C09125=1232.862,309.297,-67.480,-176.248,6.770,148.147
C09126=1232.866,309.049,-67.449,-176.251,6.767,148.147
C09127=1232.870,308.801,-67.420,-176.253,6.765,148.147
C09128=1232.875,308.552,-67.390,-176.255,6.763,148.147
C09129=1232.880,308.304,-67.361,-176.257,6.760,148.147
C09130=1232.884,308.056,-67.331,-176.260,6.757,148.147
C09131=1232.888,307.808,-67.301,-176.262,6.755,148.148
C09132=1232.892,307.560,-67.271,-176.264,6.753,148.148
C09133=1232.897,307.311,-67.241,-176.266,6.751,148.148
C09134=1232.901,307.063,-67.212,-176.269,6.748,148.148
C09135=1232.905,306.815,-67.182,-176.271,6.746,148.148
C09136=1232.909,306.566,-67.153,-176.273,6.743,148.148
C09137=1232.913,306.318,-67.124,-176.275,6.741,148.148
C09138=1232.918,306.070,-67.094,-176.278,6.739,148.148
C09139=1232.923,305.821,-67.064,-176.280,6.736,148.148
C09140=1232.926,305.574,-67.034,-176.282,6.734,148.148
C09141=1232.931,305.325,-67.004,-176.284,6.732,148.148
C09142=1232.935,305.077,-66.975,-176.286,6.729,148.148
C09143=1232.940,304.830,-66.946,-176.289,6.726,148.148
C09144=1232.944,304.581,-66.916,-176.291,6.724,148.148
C09145=1232.948,304.333,-66.887,-176.293,6.722,148.148
C09146=1232.952,304.085,-66.858,-176.295,6.720,148.148
C09147=1232.956,303.837,-66.828,-176.298,6.718,148.149
C09148=1232.960,303.588,-66.799,-176.301,6.715,148.149
C09149=1232.965,303.340,-66.769,-176.303,6.712,148.149
C09150=1232.970,303.091,-66.739,-176.305,6.710,148.149
C09151=1232.974,302.843,-66.710,-176.307,6.708,148.149
C09152=1232.979,302.595,-66.681,-176.310,6.705,148.149
C09153=1232.983,302.347,-66.652,-176.312,6.703,148.149
C09154=1232.987,302.098,-66.622,-176.314,6.700,148.149
C09155=1232.991,301.850,-66.593,-176.316,6.698,148.149
C09156=1232.996,301.602,-66.564,-176.319,6.696,148.149
C09157=1233.000,301.354,-66.534,-176.321,6.693,148.149
C09158=1233.004,301.105,-66.505,-176.323,6.691,148.149
C09159=1233.009,300.858,-66.476,-176.325,6.689,148.149
C09160=1233.013,300.610,-66.446,-176.327,6.687,148.149
C09161=1233.017,300.361,-66.417,-176.331,6.684,148.150
C09162=1233.022,300.112,-66.388,-176.333,6.682,148.150
C09163=1233.026,299.864,-66.358,-176.335,6.679,148.150
C09164=1233.031,299.617,-66.329,-176.337,6.677,148.150
C09165=1233.035,299.368,-66.300,-176.339,6.675,148.150
C09166=1233.039,299.119,-66.271,-176.342,6.672,148.150
C09167=1233.043,298.871,-66.242,-176.344,6.670,148.150
C09168=1233.047,298.623,-66.213,-176.346,6.668,148.150
C09169=1233.051,298.375,-66.183,-176.348,6.665,148.150
C09170=1233.056,298.127,-66.155,-176.351,6.663,148.150
C09171=1233.060,297.878,-66.126,-176.354,6.660,148.151
C09172=1233.064,297.630,-66.096,-176.356,6.658,148.151
C09173=1233.069,297.381,-66.067,-176.358,6.656,148.151
C09174=1233.074,297.134,-66.038,-176.360,6.654,148.151
C09175=1233.078,296.885,-66.009,-176.362,6.652,148.151
C09176=1233.082,296.637,-65.979,-176.365,6.649,148.151
C09177=1233.086,296.389,-65.951,-176.367,6.647,148.151
C09178=1233.090,296.140,-65.922,-176.369,6.644,148.151
C09179=1233.095,295.892,-65.893,-176.372,6.642,148.151
C09180=1233.099,295.644,-65.864,-176.374,6.640,148.151
C09181=1233.103,295.396,-65.834,-176.377,6.637,148.151
C09182=1233.108,295.147,-65.806,-176.379,6.635,148.152
C09183=1233.112,294.899,-65.777,-176.381,6.633,148.152
C09184=1233.116,294.651,-65.749,-176.384,6.631,148.152
C09185=1233.121,294.402,-65.719,-176.386,6.629,148.152
C09186=1233.125,294.155,-65.690,-176.388,6.626,148.152
C09187=1233.130,293.906,-65.661,-176.390,6.623,148.152
C09188=1233.133,293.658,-65.632,-176.393,6.621,148.152
C09189=1233.138,293.409,-65.604,-176.395,6.619,148.152
C09190=1233.143,293.161,-65.575,-176.397,6.617,148.152
C09191=1233.147,292.913,-65.546,-176.400,6.614,148.153
C09192=1233.151,292.665,-65.517,-176.402,6.612,148.153
C09193=1233.156,292.416,-65.489,-176.405,6.610,148.153
C09194=1233.160,292.168,-65.459,-176.407,6.608,148.153
C09195=1233.164,291.919,-65.430,-176.409,6.606,148.153
C09196=1233.169,291.671,-65.403,-176.411,6.603,148.153
C09197=1233.173,291.423,-65.373,-176.414,6.600,148.153
C09198=1233.177,291.174,-65.344,-176.417,6.598,148.153
C09199=1233.181,290.927,-65.316,-176.419,6.596,148.154
C09200=1233.186,290.678,-65.287,-176.421,6.594,148.154
C09201=1233.190,290.430,-65.258,-176.423,6.592,148.154
C09202=1233.195,290.182,-65.229,-176.426,6.590,148.154
C09203=1233.199,289.908,-65.198,-176.429,6.587,148.154
C09204=1233.204,289.633,-65.167,-176.431,6.585,148.154
C09205=1233.209,289.359,-65.135,-176.434,6.582,148.154
C09206=1233.214,289.086,-65.103,-176.436,6.580,148.155
C09207=1233.218,288.837,-65.074,-176.439,6.577,148.155
C09208=1233.222,288.588,-65.046,-176.441,6.575,148.155
C09209=1233.227,288.341,-65.017,-176.443,6.573,148.155
C09210=1233.231,288.092,-64.988,-176.445,6.571,148.155
C09211=1233.235,287.843,-64.960,-176.448,6.569,148.155
C09212=1233.240,287.595,-64.932,-176.450,6.566,148.155
C09213=1233.244,287.347,-64.903,-176.453,6.564,148.156
C09214=1233.249,287.099,-64.875,-176.455,6.561,148.156
C09215=1233.253,286.850,-64.846,-176.457,6.559,148.156
C09216=1233.257,286.602,-64.818,-176.460,6.557,148.156
C09217=1233.262,286.353,-64.789,-176.462,6.555,148.156
C09218=1233.266,286.105,-64.760,-176.465,6.553,148.156
C09219=1233.271,285.857,-64.732,-176.467,6.550,148.156
C09220=1233.274,285.609,-64.704,-176.470,6.548,148.156
C09221=1233.280,285.360,-64.676,-176.472,6.546,148.157
C09222=1233.283,285.112,-64.647,-176.474,6.544,148.157
C09223=1233.288,284.864,-64.619,-176.477,6.542,148.157
C09224=1233.293,284.615,-64.590,-176.479,6.540,148.157
C09225=1233.296,284.367,-64.562,-176.481,6.537,148.157
C09226=1233.301,284.119,-64.533,-176.484,6.535,148.157
C09227=1233.305,283.870,-64.505,-176.486,6.532,148.157
C09228=1233.310,283.622,-64.477,-176.489,6.531,148.158
C09229=1233.314,283.373,-64.448,-176.491,6.528,148.158
C09230=1233.318,283.125,-64.421,-176.494,6.526,148.158
C09231=1233.323,282.877,-64.392,-176.496,6.524,148.158
C09232=1233.327,282.629,-64.364,-176.498,6.522,148.158
C09233=1233.332,282.380,-64.335,-176.501,6.519,148.158
C09234=1233.336,282.132,-64.308,-176.503,6.517,148.158
C09235=1233.340,281.883,-64.279,-176.506,6.515,148.159
C09236=1233.345,281.635,-64.251,-176.508,6.513,148.159
C09237=1233.349,281.386,-64.222,-176.510,6.511,148.159
C09238=1233.354,281.138,-64.195,-176.512,6.509,148.159
C09239=1233.357,280.890,-64.166,-176.515,6.507,148.159
C09240=1233.363,280.642,-64.138,-176.517,6.505,148.160
C09241=1233.366,280.393,-64.110,-176.520,6.502,148.160
C09242=1233.371,280.145,-64.082,-176.522,6.500,148.160
C09243=1233.375,279.896,-64.053,-176.525,6.498,148.160
C09244=1233.379,279.648,-64.026,-176.527,6.496,148.160
C09245=1233.384,279.400,-63.997,-176.530,6.494,148.161
C09246=1233.389,279.151,-63.970,-176.532,6.491,148.161
C09247=1233.392,278.902,-63.942,-176.534,6.489,148.161
C09248=1233.397,278.654,-63.913,-176.536,6.487,148.161
C09249=1233.402,278.406,-63.886,-176.539,6.485,148.161
C09250=1233.406,278.158,-63.857,-176.542,6.482,148.161
C09251=1233.411,277.910,-63.829,-176.544,6.480,148.161
C09252=1233.414,277.661,-63.801,-176.546,6.478,148.162
C09253=1233.419,277.413,-63.774,-176.549,6.476,148.162
C09254=1233.424,277.164,-63.745,-176.551,6.474,148.162
C09255=1233.428,276.916,-63.717,-176.554,6.472,148.162
C09256=1233.432,276.668,-63.690,-176.556,6.470,148.162
C09257=1233.436,276.419,-63.662,-176.558,6.468,148.163
C09258=1233.441,276.171,-63.634,-176.561,6.466,148.163
C09259=1233.445,275.922,-63.606,-176.564,6.463,148.163
C09260=1233.449,275.674,-63.578,-176.566,6.461,148.163
C09261=1233.454,275.426,-63.551,-176.568,6.459,148.163
C09262=1233.459,275.177,-63.522,-176.571,6.457,148.163
C09263=1233.463,274.929,-63.494,-176.573,6.455,148.164
C09264=1233.467,274.680,-63.467,-176.575,6.453,148.164
C09265=1233.471,274.432,-63.439,-176.578,6.451,148.164
C09266=1233.476,274.184,-63.411,-176.580,6.449,148.164
C09267=1233.480,273.934,-63.383,-176.583,6.447,148.164
C09268=1233.485,273.687,-63.356,-176.585,6.445,148.165
C09269=1233.489,273.439,-63.328,-176.588,6.442,148.165
C09270=1233.493,273.189,-63.300,-176.590,6.440,148.165
C09271=1233.498,272.941,-63.272,-176.592,6.438,148.165
C09272=1233.503,272.693,-63.245,-176.595,6.436,148.165
C09273=1233.507,272.444,-63.217,-176.597,6.433,148.165
C09274=1233.511,272.196,-63.189,-176.600,6.432,148.166
C09275=1233.516,271.948,-63.162,-176.602,6.430,148.166
C09276=1233.520,271.699,-63.134,-176.604,6.427,148.166
C09277=1233.524,271.451,-63.107,-176.607,6.426,148.166
C09278=1233.529,271.203,-63.078,-176.609,6.423,148.166
C09279=1233.533,270.953,-63.051,-176.612,6.421,148.167
C09280=1233.538,270.705,-63.023,-176.614,6.419,148.167
C09281=1233.542,270.457,-62.996,-176.617,6.417,148.167
C09282=1233.546,270.208,-62.968,-176.620,6.415,148.167
C09283=1233.551,269.960,-62.941,-176.622,6.412,148.167
C09284=1233.555,269.712,-62.913,-176.624,6.410,148.168
C09285=1233.559,269.463,-62.886,-176.626,6.408,148.168
C09286=1233.564,269.214,-62.859,-176.629,6.406,148.168
C09287=1233.568,268.966,-62.831,-176.632,6.404,148.168
C09288=1233.573,268.718,-62.804,-176.634,6.402,148.168
C09289=1233.577,268.469,-62.776,-176.636,6.400,148.169
C09290=1233.581,268.221,-62.749,-176.639,6.398,148.169
C09291=1233.586,267.973,-62.721,-176.641,6.396,148.169
C09292=1233.591,267.724,-62.693,-176.644,6.394,148.169
C09293=1233.595,267.475,-62.666,-176.646,6.392,148.169
C09294=1233.599,267.227,-62.638,-176.648,6.390,148.170
C09295=1233.604,266.979,-62.611,-176.651,6.388,148.170
C09296=1233.609,266.730,-62.584,-176.653,6.386,148.170
C09297=1233.612,266.482,-62.556,-176.656,6.384,148.170
C09298=1233.617,266.233,-62.529,-176.658,6.382,148.171
C09299=1233.621,265.985,-62.502,-176.660,6.380,148.171
C09300=1233.626,265.736,-62.475,-176.664,6.377,148.171
C09301=1233.630,265.489,-62.447,-176.666,6.375,148.171
C09302=1233.634,265.239,-62.420,-176.668,6.373,148.171
C09303=1233.639,264.991,-62.393,-176.671,6.371,148.172
C09304=1233.643,264.742,-62.366,-176.673,6.369,148.172
C09305=1233.648,264.494,-62.338,-176.676,6.367,148.172
C09306=1233.652,264.246,-62.311,-176.678,6.365,148.172
C09307=1233.657,263.973,-62.280,-176.681,6.363,148.173
C09308=1233.662,263.700,-62.251,-176.683,6.361,148.173
C09309=1233.666,263.427,-62.221,-176.686,6.358,148.173
C09310=1233.672,263.155,-62.191,-176.689,6.357,148.173
C09311=1233.676,262.906,-62.164,-176.691,6.355,148.174
C09312=1233.680,262.658,-62.138,-176.693,6.352,148.174
C09313=1233.685,262.410,-62.110,-176.696,6.351,148.174
C09314=1233.689,262.162,-62.083,-176.699,6.349,148.174
C09315=1233.693,261.913,-62.055,-176.701,6.347,148.175
C09316=1233.698,261.664,-62.028,-176.703,6.345,148.175
C09317=1233.703,261.416,-62.001,-176.706,6.343,148.175
C09318=1233.707,261.167,-61.974,-176.709,6.341,148.175
C09319=1233.711,260.919,-61.948,-176.711,6.339,148.175
C09320=1233.716,260.670,-61.921,-176.713,6.337,148.176
C09321=1233.720,260.422,-61.894,-176.716,6.335,148.176
C09322=1233.725,260.173,-61.867,-176.718,6.333,148.176
C09323=1233.729,259.924,-61.839,-176.721,6.331,148.176
C09324=1233.733,259.676,-61.813,-176.723,6.329,148.177
C09325=1233.738,259.427,-61.786,-176.726,6.327,148.177
C09326=1233.742,259.179,-61.759,-176.728,6.325,148.177
C09327=1233.747,258.931,-61.731,-176.730,6.323,148.177
C09328=1233.751,258.682,-61.705,-176.733,6.321,148.178
C09329=1233.756,258.434,-61.678,-176.735,6.319,148.178
C09330=1233.760,258.185,-61.651,-176.738,6.317,148.178
C09331=1233.765,257.937,-61.624,-176.740,6.315,148.178
C09332=1233.769,257.689,-61.597,-176.743,6.313,148.179
C09333=1233.773,257.439,-61.570,-176.745,6.311,148.179
C09334=1233.778,257.191,-61.543,-176.748,6.309,148.179
C09335=1233.782,256.942,-61.516,-176.750,6.307,148.179
C09336=1233.786,256.694,-61.489,-176.753,6.305,148.180
C09337=1233.791,256.445,-61.463,-176.755,6.303,148.180
C09338=1233.796,256.197,-61.436,-176.758,6.301,148.180
C09339=1233.800,255.948,-61.409,-176.760,6.299,148.180
C09340=1233.804,255.700,-61.382,-176.763,6.297,148.181
C09341=1233.809,255.451,-61.355,-176.765,6.295,148.181
C09342=1233.813,255.203,-61.329,-176.768,6.293,148.181
C09343=1233.818,254.954,-61.303,-176.770,6.291,148.181
C09344=1233.823,254.706,-61.275,-176.773,6.289,148.182
C09345=1233.827,254.458,-61.249,-176.775,6.287,148.182
C09346=1233.831,254.209,-61.222,-176.778,6.285,148.182
C09347=1233.836,253.960,-61.196,-176.780,6.283,148.182
C09348=1233.840,253.712,-61.169,-176.783,6.281,148.183
C09349=1233.845,253.463,-61.142,-176.785,6.279,148.183
C09350=1233.849,253.215,-61.116,-176.787,6.277,148.183
C09351=1233.854,252.966,-61.089,-176.790,6.275,148.183
C09352=1233.858,252.717,-61.062,-176.793,6.274,148.184
C09353=1233.862,252.469,-61.036,-176.795,6.271,148.184
C09354=1233.867,252.221,-61.009,-176.797,6.269,148.184
C09355=1233.871,251.972,-60.983,-176.800,6.268,148.184
C09356=1233.876,251.723,-60.956,-176.803,6.266,148.185
C09357=1233.880,251.475,-60.929,-176.805,6.264,148.185
C09358=1233.885,251.226,-60.903,-176.807,6.262,148.185
C09359=1233.888,250.978,-60.877,-176.810,6.260,148.185
C09360=1233.893,250.729,-60.850,-176.813,6.258,148.186
C09361=1233.897,250.481,-60.824,-176.815,6.256,148.186
C09362=1233.902,250.232,-60.797,-176.818,6.254,148.186
C09363=1233.906,249.983,-60.771,-176.820,6.252,148.186
C09364=1233.911,249.735,-60.744,-176.822,6.250,148.187
C09365=1233.915,249.486,-60.718,-176.825,6.249,148.187
C09366=1233.920,249.238,-60.691,-176.827,6.247,148.187
C09367=1233.925,248.989,-60.666,-176.830,6.245,148.188
C09368=1233.929,248.741,-60.639,-176.832,6.243,148.188
C09369=1233.934,248.492,-60.613,-176.834,6.241,148.188
C09370=1233.938,248.244,-60.586,-176.837,6.239,148.188
C09371=1233.942,247.995,-60.560,-176.840,6.237,148.189
C09372=1233.947,247.746,-60.533,-176.842,6.235,148.189
C09373=1233.951,247.498,-60.507,-176.844,6.233,148.189
C09374=1233.956,247.249,-60.480,-176.847,6.231,148.189
C09375=1233.960,247.000,-60.454,-176.850,6.229,148.190
C09376=1233.964,246.752,-60.428,-176.852,6.227,148.190
C09377=1233.970,246.504,-60.402,-176.855,6.226,148.190
C09378=1233.974,246.255,-60.376,-176.857,6.224,148.191
C09379=1233.979,246.006,-60.349,-176.860,6.221,148.191
C09380=1233.982,245.758,-60.323,-176.862,6.220,148.191
C09381=1233.987,245.509,-60.297,-176.865,6.218,148.191
C09382=1233.992,245.260,-60.271,-176.867,6.217,148.192
C09383=1233.996,245.012,-60.244,-176.869,6.215,148.192
C09384=1234.000,244.764,-60.219,-176.872,6.213,148.192
C09385=1234.005,244.515,-60.192,-176.875,6.211,148.193
C09386=1234.009,244.267,-60.166,-176.877,6.209,148.193
C09387=1234.013,244.018,-60.140,-176.879,6.207,148.193
C09388=1234.018,243.769,-60.114,-176.882,6.205,148.193
C09389=1234.022,243.521,-60.087,-176.885,6.203,148.194
C09390=1234.027,243.272,-60.062,-176.887,6.201,148.194
C09391=1234.032,243.023,-60.036,-176.890,6.199,148.194
C09392=1234.036,242.775,-60.009,-176.892,6.197,148.194
C09393=1234.040,242.526,-59.983,-176.895,6.195,148.195
C09394=1234.045,242.277,-59.957,-176.897,6.194,148.195
C09395=1234.049,242.028,-59.931,-176.899,6.192,148.195
C09396=1234.054,241.780,-59.906,-176.902,6.190,148.196
C09397=1234.058,241.532,-59.879,-176.905,6.189,148.196
C09398=1234.063,241.283,-59.853,-176.907,6.187,148.196
C09399=1234.067,241.034,-59.827,-176.910,6.185,148.196
C09400=1234.072,240.785,-59.802,-176.912,6.183,148.197
C09401=1234.076,240.537,-59.776,-176.914,6.181,148.197
C09402=1234.081,240.289,-59.749,-176.917,6.179,148.197
C09403=1234.085,240.040,-59.723,-176.920,6.177,148.198
C09404=1234.090,239.791,-59.698,-176.922,6.175,148.198
C09405=1234.094,239.543,-59.672,-176.924,6.174,148.198
C09406=1234.099,239.294,-59.646,-176.927,6.172,148.199
C09407=1234.104,239.045,-59.620,-176.930,6.170,148.199
C09408=1234.108,238.796,-59.594,-176.932,6.168,148.199
C09409=1234.112,238.549,-59.568,-176.934,6.166,148.199
C09410=1234.117,238.300,-59.543,-176.937,6.164,148.200
C09411=1234.121,238.028,-59.515,-176.940,6.162,148.200
C09412=1234.127,237.757,-59.487,-176.943,6.161,148.200
C09413=1234.131,237.486,-59.458,-176.945,6.159,148.201
C09414=1234.136,237.215,-59.430,-176.948,6.156,148.201
C09415=1234.141,236.965,-59.404,-176.951,6.155,148.201
C09416=1234.145,236.717,-59.378,-176.953,6.153,148.202
C09417=1234.150,236.469,-59.353,-176.955,6.151,148.202
C09418=1234.154,236.220,-59.327,-176.958,6.149,148.202
C09419=1234.159,235.971,-59.301,-176.960,6.147,148.202
C09420=1234.163,235.722,-59.276,-176.963,6.145,148.203
C09421=1234.168,235.474,-59.250,-176.966,6.143,148.203
C09422=1234.172,235.225,-59.225,-176.968,6.142,148.203
C09423=1234.176,234.976,-59.199,-176.970,6.141,148.204
C09424=1234.181,234.728,-59.173,-176.973,6.139,148.204
C09425=1234.186,234.479,-59.147,-176.976,6.137,148.204
C09426=1234.190,234.230,-59.122,-176.978,6.135,148.205
C09427=1234.195,233.982,-59.097,-176.981,6.133,148.205
C09428=1234.200,233.733,-59.071,-176.983,6.131,148.205
C09429=1234.204,233.484,-59.045,-176.986,6.129,148.206
C09430=1234.209,233.236,-59.020,-176.989,6.127,148.206
C09431=1234.213,232.987,-58.994,-176.990,6.126,148.206
C09432=1234.217,232.738,-58.968,-176.993,6.124,148.206
C09433=1234.222,232.490,-58.944,-176.996,6.122,148.207
C09434=1234.226,232.241,-58.918,-176.998,6.120,148.207
C09435=1234.231,231.993,-58.893,-177.001,6.119,148.207
C09436=1234.235,231.744,-58.867,-177.003,6.117,148.208
C09437=1234.240,231.495,-58.841,-177.006,6.115,148.208
C09438=1234.245,231.246,-58.816,-177.008,6.114,148.208
C09439=1234.249,230.998,-58.791,-177.011,6.112,148.209
C09440=1234.254,230.749,-58.765,-177.013,6.110,148.209
C09441=1234.258,230.501,-58.739,-177.016,6.108,148.209
C09442=1234.262,230.252,-58.715,-177.019,6.106,148.210
C09443=1234.267,230.003,-58.690,-177.021,6.104,148.210
C09444=1234.271,229.755,-58.664,-177.024,6.102,148.210
C09445=1234.276,229.507,-58.638,-177.026,6.101,148.211
C09446=1234.280,229.257,-58.613,-177.028,6.100,148.211
C09447=1234.285,229.008,-58.588,-177.031,6.098,148.211
C09448=1234.289,228.760,-58.562,-177.034,6.096,148.212
C09449=1234.294,228.511,-58.537,-177.036,6.094,148.212
C09450=1234.299,228.263,-58.512,-177.039,6.092,148.212
C09451=1234.303,228.014,-58.486,-177.041,6.091,148.213
C09452=1234.308,227.765,-58.461,-177.044,6.089,148.213
C09453=1234.312,227.517,-58.436,-177.046,6.087,148.213
C09454=1234.316,227.267,-58.411,-177.049,6.085,148.214
C09455=1234.321,227.019,-58.386,-177.051,6.083,148.214
C09456=1234.325,226.770,-58.360,-177.054,6.082,148.214
C09457=1234.330,226.522,-58.335,-177.057,6.080,148.214
C09458=1234.334,226.273,-58.310,-177.059,6.079,148.215
C09459=1234.339,226.024,-58.286,-177.061,6.077,148.215
C09460=1234.343,225.776,-58.260,-177.064,6.075,148.216
C09461=1234.348,225.527,-58.235,-177.067,6.073,148.216
C09462=1234.352,225.278,-58.209,-177.069,6.071,148.216
C09463=1234.358,225.029,-58.185,-177.072,6.069,148.216
C09464=1234.361,224.781,-58.160,-177.074,6.068,148.217
C09465=1234.366,224.532,-58.135,-177.077,6.066,148.217
C09466=1234.370,224.283,-58.109,-177.079,6.064,148.217
C09467=1234.376,224.035,-58.085,-177.082,6.063,148.218
C09468=1234.379,223.786,-58.059,-177.084,6.061,148.218
C09469=1234.384,223.537,-58.035,-177.086,6.060,148.218
C09470=1234.388,223.289,-58.009,-177.089,6.058,148.219
C09471=1234.394,223.040,-57.984,-177.092,6.056,148.219
C09472=1234.397,222.791,-57.959,-177.094,6.054,148.219
C09473=1234.402,222.543,-57.934,-177.097,6.052,148.220
C09474=1234.407,222.294,-57.910,-177.100,6.050,148.220
C09475=1234.411,222.045,-57.884,-177.102,6.049,148.220
C09476=1234.416,221.797,-57.860,-177.104,6.047,148.221
C09477=1234.420,221.547,-57.835,-177.107,6.046,148.221
C09478=1234.425,221.299,-57.810,-177.110,6.044,148.221
C09479=1234.429,221.050,-57.785,-177.112,6.042,148.222
C09480=1234.434,220.802,-57.760,-177.114,6.041,148.222
C09481=1234.438,220.552,-57.735,-177.117,6.039,148.222
C09482=1234.443,220.304,-57.711,-177.119,6.037,148.223
C09483=1234.448,220.055,-57.686,-177.122,6.035,148.223
C09484=1234.452,219.807,-57.660,-177.125,6.033,148.223
C09485=1234.457,219.558,-57.636,-177.127,6.031,148.224
C09486=1234.461,219.309,-57.611,-177.129,6.030,148.224
C09487=1234.465,219.061,-57.586,-177.132,6.028,148.224
C09488=1234.470,218.812,-57.562,-177.135,6.027,148.225
C09489=1234.475,218.563,-57.537,-177.138,6.025,148.225
C09490=1234.479,218.314,-57.513,-177.140,6.023,148.226
C09491=1234.484,218.065,-57.488,-177.142,6.022,148.226
C09492=1234.488,217.817,-57.463,-177.145,6.020,148.226
C09493=1234.493,217.568,-57.438,-177.148,6.018,148.227
C09494=1234.498,217.319,-57.413,-177.150,6.017,148.227
C09495=1234.502,217.071,-57.389,-177.153,6.015,148.227
C09496=1234.506,216.821,-57.364,-177.155,6.014,148.228
C09497=1234.511,216.573,-57.339,-177.158,6.012,148.228
C09498=1234.516,216.325,-57.314,-177.160,6.010,148.228
C09499=1234.519,216.076,-57.290,-177.163,6.008,148.229
C09500=1234.525,215.827,-57.265,-177.166,6.006,148.229
C09501=1234.529,215.578,-57.241,-177.168,6.005,148.229
C09502=1234.533,215.329,-57.216,-177.170,6.003,148.230
C09503=1234.538,215.081,-57.192,-177.173,6.002,148.230
C09504=1234.543,214.832,-57.167,-177.176,6.000,148.231
C09505=1234.547,214.583,-57.143,-177.179,5.998,148.231
C09506=1234.552,214.334,-57.118,-177.181,5.997,148.231
C09507=1234.556,214.086,-57.094,-177.183,5.995,148.232
C09508=1234.561,213.837,-57.069,-177.186,5.993,148.232
C09509=1234.565,213.588,-57.044,-177.189,5.991,148.232
C09510=1234.570,213.340,-57.020,-177.191,5.990,148.233
C09511=1234.574,213.091,-56.996,-177.193,5.988,148.233
C09512=1234.579,212.842,-56.971,-177.196,5.987,148.233
C09513=1234.583,212.593,-56.947,-177.198,5.985,148.234
C09514=1234.589,212.345,-56.922,-177.202,5.983,148.234
C09515=1234.593,212.073,-56.896,-177.204,5.981,148.235
C09516=1234.598,211.803,-56.869,-177.207,5.979,148.235
C09517=1234.603,211.533,-56.843,-177.209,5.978,148.235
C09518=1234.608,211.263,-56.816,-177.213,5.976,148.236
C09519=1234.613,211.014,-56.793,-177.215,5.975,148.236
C09520=1234.617,210.764,-56.768,-177.217,5.973,148.236
C09521=1234.622,210.516,-56.744,-177.220,5.971,148.237
C09522=1234.626,210.268,-56.720,-177.223,5.969,148.237
C09523=1234.631,210.019,-56.695,-177.225,5.968,148.238
C09524=1234.635,209.770,-56.670,-177.227,5.966,148.238
C09525=1234.640,209.521,-56.646,-177.230,5.965,148.238
C09526=1234.645,209.273,-56.622,-177.233,5.963,148.239
C09527=1234.649,209.024,-56.598,-177.235,5.962,148.239
C09528=1234.654,208.774,-56.573,-177.238,5.960,148.239
C09529=1234.658,208.526,-56.549,-177.240,5.958,148.240
C09530=1234.663,208.277,-56.525,-177.243,5.956,148.240
C09531=1234.668,208.029,-56.500,-177.245,5.955,148.240
C09532=1234.672,207.780,-56.477,-177.248,5.954,148.241
C09533=1234.676,207.531,-56.453,-177.251,5.952,148.241
C09534=1234.681,207.282,-56.429,-177.253,5.950,148.242
C09535=1234.686,207.033,-56.404,-177.255,5.949,148.242
C09536=1234.690,206.784,-56.381,-177.258,5.947,148.242
C09537=1234.695,206.536,-56.356,-177.261,5.945,148.243
C09538=1234.699,206.287,-56.331,-177.263,5.944,148.243
C09539=1234.704,206.038,-56.307,-177.265,5.942,148.243
C09540=1234.708,205.789,-56.284,-177.268,5.941,148.244
C09541=1234.713,205.541,-56.260,-177.271,5.939,148.244
C09542=1234.718,205.292,-56.235,-177.273,5.938,148.245
C09543=1234.723,205.043,-56.212,-177.276,5.936,148.245
C09544=1234.726,204.794,-56.187,-177.279,5.934,148.245
C09545=1234.731,204.545,-56.163,-177.281,5.932,148.246
C09546=1234.736,204.296,-56.140,-177.283,5.931,148.246
C09547=1234.741,204.048,-56.115,-177.286,5.930,148.246
C09548=1234.745,203.799,-56.092,-177.289,5.928,148.247
C09549=1234.750,203.550,-56.068,-177.291,5.927,148.247
C09550=1234.754,203.302,-56.044,-177.294,5.925,148.248
C09551=1234.758,203.052,-56.020,-177.296,5.923,148.248
C09552=1234.763,202.804,-55.996,-177.299,5.921,148.248
C09553=1234.768,202.554,-55.972,-177.301,5.920,148.249
C09554=1234.773,202.306,-55.948,-177.304,5.919,148.249
C09555=1234.777,202.057,-55.924,-177.307,5.917,148.250
C09556=1234.782,201.808,-55.901,-177.309,5.916,148.250
C09557=1234.786,201.560,-55.877,-177.312,5.914,148.250
C09558=1234.791,201.311,-55.853,-177.314,5.912,148.251
C09559=1234.795,201.063,-55.829,-177.316,5.911,148.251
C09560=1234.800,200.813,-55.805,-177.319,5.910,148.252
C09561=1234.804,200.564,-55.781,-177.322,5.908,148.252
C09562=1234.809,200.315,-55.757,-177.325,5.906,148.252
C09563=1234.814,200.066,-55.734,-177.327,5.905,148.253
C09564=1234.818,199.818,-55.710,-177.329,5.903,148.253
C09565=1234.823,199.569,-55.687,-177.332,5.901,148.253
C09566=1234.827,199.320,-55.662,-177.335,5.900,148.254
C09567=1234.832,199.071,-55.639,-177.337,5.899,148.254
C09568=1234.836,198.823,-55.615,-177.340,5.897,148.255
C09569=1234.841,198.574,-55.592,-177.342,5.896,148.255
C09570=1234.846,198.325,-55.568,-177.345,5.894,148.255
C09571=1234.850,198.076,-55.544,-177.348,5.892,148.256
C09572=1234.855,197.827,-55.521,-177.350,5.891,148.256
C09573=1234.859,197.579,-55.497,-177.352,5.889,148.257
C09574=1234.864,197.330,-55.473,-177.355,5.888,148.257
C09575=1234.869,197.081,-55.450,-177.357,5.887,148.257
C09576=1234.873,196.832,-55.426,-177.360,5.885,148.258
C09577=1234.878,196.583,-55.403,-177.363,5.883,148.258
C09578=1234.882,196.334,-55.379,-177.365,5.882,148.259
C09579=1234.887,196.085,-55.356,-177.368,5.880,148.259
C09580=1234.891,195.837,-55.332,-177.370,5.878,148.259
C09581=1234.896,195.588,-55.308,-177.373,5.878,148.260
C09582=1234.901,195.339,-55.285,-177.375,5.876,148.260
C09583=1234.905,195.090,-55.261,-177.378,5.874,148.261
C09584=1234.910,194.841,-55.238,-177.380,5.873,148.261
C09585=1234.915,194.592,-55.214,-177.383,5.871,148.261
C09586=1234.919,194.343,-55.191,-177.386,5.870,148.262
C09587=1234.924,194.094,-55.168,-177.388,5.869,148.262
C09588=1234.928,193.846,-55.144,-177.391,5.867,148.263
C09589=1234.933,193.597,-55.120,-177.393,5.865,148.263
C09590=1234.938,193.348,-55.097,-177.395,5.864,148.263
C09591=1234.943,193.099,-55.073,-177.398,5.862,148.264
C09592=1234.947,192.850,-55.050,-177.401,5.860,148.264
C09593=1234.951,192.602,-55.027,-177.403,5.859,148.265
C09594=1234.956,192.353,-55.003,-177.406,5.858,148.265
C09595=1234.960,192.104,-54.980,-177.408,5.857,148.265
C09596=1234.965,191.855,-54.957,-177.411,5.855,148.266
C09597=1234.970,191.605,-54.933,-177.414,5.853,148.266
C09598=1234.974,191.356,-54.910,-177.416,5.852,148.267
C09599=1234.979,191.107,-54.886,-177.418,5.850,148.267
C09600=1234.984,190.859,-54.864,-177.422,5.849,148.268
C09601=1234.988,190.610,-54.841,-177.424,5.848,148.268
C09602=1234.993,190.361,-54.817,-177.426,5.846,148.268
C09603=1234.997,190.113,-54.793,-177.428,5.845,148.269
C09604=1235.002,189.864,-54.770,-177.431,5.843,148.269
C09605=1235.007,189.615,-54.747,-177.434,5.842,148.270
C09606=1235.011,189.366,-54.724,-177.436,5.840,148.270
C09607=1235.016,189.117,-54.700,-177.439,5.839,148.270
C09608=1235.020,188.868,-54.677,-177.442,5.837,148.271
C09609=1235.026,188.620,-54.654,-177.444,5.836,148.271
C09610=1235.030,188.371,-54.631,-177.447,5.834,148.272
C09611=1235.034,188.122,-54.608,-177.449,5.833,148.272
C09612=1235.039,187.873,-54.585,-177.451,5.831,148.272
C09613=1235.044,187.623,-54.562,-177.455,5.830,148.273
C09614=1235.048,187.375,-54.539,-177.457,5.829,148.273
C09615=1235.053,187.126,-54.516,-177.459,5.827,148.274
C09616=1235.058,186.877,-54.493,-177.461,5.826,148.274
C09617=1235.063,186.628,-54.469,-177.464,5.824,148.275
C09618=1235.067,186.379,-54.447,-177.467,5.823,148.275
C09619=1235.072,186.110,-54.422,-177.469,5.822,148.275
C09620=1235.077,185.840,-54.397,-177.472,5.820,148.276
C09621=1235.082,185.570,-54.372,-177.475,5.818,148.276
C09622=1235.087,185.301,-54.347,-177.478,5.817,148.277
C09623=1235.092,185.052,-54.324,-177.481,5.815,148.277
C09624=1235.096,184.803,-54.301,-177.483,5.814,148.278
C09625=1235.100,184.554,-54.278,-177.486,5.812,148.278
C09626=1235.105,184.305,-54.254,-177.488,5.811,148.279
C09627=1235.109,184.056,-54.232,-177.491,5.809,148.279
C09628=1235.115,183.807,-54.209,-177.493,5.808,148.279
C09629=1235.119,183.558,-54.186,-177.496,5.807,148.280
C09630=1235.123,183.309,-54.163,-177.499,5.805,148.280
C09631=1235.128,183.060,-54.140,-177.501,5.804,148.281
C09632=1235.133,182.812,-54.117,-177.504,5.802,148.281
C09633=1235.138,182.563,-54.095,-177.506,5.801,148.282
C09634=1235.142,182.314,-54.071,-177.509,5.800,148.282
C09635=1235.146,182.065,-54.049,-177.511,5.798,148.282
C09636=1235.151,181.815,-54.026,-177.514,5.797,148.283
C09637=1235.156,181.567,-54.004,-177.516,5.795,148.283
C09638=1235.161,181.318,-53.980,-177.518,5.794,148.284
C09639=1235.165,181.069,-53.957,-177.521,5.792,148.284
C09640=1235.170,180.820,-53.935,-177.524,5.792,148.285
C09641=1235.175,180.572,-53.912,-177.526,5.790,148.285
C09642=1235.179,180.323,-53.889,-177.528,5.789,148.285
C09643=1235.184,180.073,-53.866,-177.532,5.787,148.286
C09644=1235.188,179.824,-53.844,-177.534,5.785,148.286
C09645=1235.193,179.576,-53.821,-177.536,5.784,148.287
C09646=1235.197,179.327,-53.799,-177.539,5.783,148.287
C09647=1235.202,179.078,-53.775,-177.542,5.782,148.288
C09648=1235.207,178.829,-53.754,-177.544,5.780,148.288
C09649=1235.212,178.580,-53.730,-177.546,5.779,148.288
C09650=1235.216,178.331,-53.708,-177.549,5.778,148.289
C09651=1235.221,178.082,-53.685,-177.551,5.777,148.289
C09652=1235.225,177.834,-53.662,-177.554,5.775,148.290
C09653=1235.230,177.584,-53.640,-177.557,5.773,148.290
C09654=1235.234,177.335,-53.617,-177.559,5.772,148.291
C09655=1235.240,177.086,-53.595,-177.562,5.770,148.291
C09656=1235.244,176.838,-53.572,-177.565,5.770,148.292
C09657=1235.249,176.588,-53.549,-177.567,5.768,148.292
C09658=1235.253,176.340,-53.527,-177.569,5.767,148.292
C09659=1235.258,176.090,-53.504,-177.572,5.765,148.293
C09660=1235.262,175.842,-53.482,-177.575,5.764,148.293
C09661=1235.267,175.593,-53.460,-177.577,5.762,148.294
C09662=1235.272,175.344,-53.437,-177.580,5.762,148.294
C09663=1235.276,175.095,-53.414,-177.582,5.760,148.295
C09664=1235.281,174.846,-53.391,-177.585,5.759,148.295
C09665=1235.286,174.597,-53.369,-177.587,5.757,148.295
C09666=1235.290,174.348,-53.347,-177.590,5.755,148.296
C09667=1235.295,174.099,-53.324,-177.592,5.754,148.296
C09668=1235.299,173.850,-53.302,-177.595,5.753,148.297
C09669=1235.305,173.602,-53.279,-177.598,5.752,148.297
C09670=1235.309,173.352,-53.257,-177.600,5.750,148.298
C09671=1235.313,173.103,-53.235,-177.602,5.749,148.298
C09672=1235.319,172.855,-53.212,-177.606,5.748,148.299
C09673=1235.323,172.605,-53.190,-177.608,5.747,148.299
C09674=1235.328,172.357,-53.169,-177.610,5.745,148.299
C09675=1235.332,172.108,-53.145,-177.613,5.744,148.300
C09676=1235.337,171.858,-53.123,-177.615,5.742,148.300
C09677=1235.342,171.610,-53.101,-177.618,5.742,148.301
C09678=1235.346,171.361,-53.078,-177.621,5.740,148.301
C09679=1235.351,171.112,-53.056,-177.623,5.739,148.302
C09680=1235.355,170.863,-53.034,-177.626,5.737,148.302
C09681=1235.360,170.613,-53.012,-177.628,5.736,148.303
C09682=1235.365,170.365,-52.989,-177.631,5.734,148.303
C09683=1235.369,170.116,-52.967,-177.633,5.734,148.304
C09684=1235.374,169.867,-52.946,-177.636,5.732,148.304
C09685=1235.379,169.617,-52.923,-177.638,5.731,148.304
C09686=1235.384,169.369,-52.901,-177.641,5.729,148.305
C09687=1235.388,169.120,-52.878,-177.643,5.728,148.305
C09688=1235.393,168.871,-52.857,-177.646,5.726,148.306
C09689=1235.398,168.622,-52.834,-177.648,5.726,148.306
C09690=1235.402,168.372,-52.812,-177.651,5.724,148.307
C09691=1235.407,168.124,-52.790,-177.653,5.723,148.307
C09692=1235.411,167.875,-52.768,-177.656,5.721,148.308
C09693=1235.417,167.626,-52.745,-177.658,5.720,148.308
C09694=1235.421,167.377,-52.723,-177.662,5.719,148.309
C09695=1235.426,167.128,-52.702,-177.664,5.718,148.309
C09696=1235.430,166.879,-52.680,-177.666,5.716,148.309
C09697=1235.435,166.631,-52.657,-177.669,5.715,148.310
C09698=1235.439,166.381,-52.635,-177.672,5.714,148.310
C09699=1235.444,166.132,-52.613,-177.674,5.712,148.311
C09700=1235.449,165.883,-52.591,-177.676,5.712,148.311
C09701=1235.454,165.634,-52.569,-177.679,5.710,148.312
C09702=1235.458,165.385,-52.547,-177.682,5.709,148.312
C09703=1235.463,165.136,-52.525,-177.684,5.707,148.313
C09704=1235.467,164.887,-52.503,-177.686,5.706,148.313
C09705=1235.473,164.638,-52.481,-177.689,5.705,148.314
C09706=1235.477,164.389,-52.459,-177.692,5.704,148.314
C09707=1235.482,164.140,-52.437,-177.695,5.702,148.315
C09708=1235.486,163.891,-52.415,-177.697,5.701,148.315
C09709=1235.491,163.642,-52.394,-177.699,5.700,148.315
C09710=1235.496,163.393,-52.372,-177.702,5.699,148.316
C09711=1235.500,163.144,-52.350,-177.705,5.697,148.316
C09712=1235.505,162.895,-52.328,-177.707,5.696,148.317
C09713=1235.509,162.646,-52.306,-177.709,5.695,148.317
C09714=1235.514,162.398,-52.284,-177.712,5.694,148.318
C09715=1235.518,162.148,-52.262,-177.715,5.693,148.318
C09716=1235.524,161.899,-52.240,-177.717,5.691,148.319
C09717=1235.528,161.650,-52.218,-177.719,5.690,148.319
C09718=1235.533,161.401,-52.196,-177.722,5.689,148.320
C09719=1235.538,161.153,-52.175,-177.725,5.688,148.320
C09720=1235.542,160.903,-52.153,-177.728,5.686,148.321
C09721=1235.547,160.654,-52.132,-177.730,5.685,148.321
C09722=1235.552,160.405,-52.110,-177.732,5.684,148.322
C09723=1235.556,160.136,-52.086,-177.735,5.683,148.322
C09724=1235.561,159.867,-52.063,-177.738,5.681,148.323
C09725=1235.567,159.597,-52.039,-177.740,5.680,148.323
C09726=1235.571,159.329,-52.016,-177.743,5.679,148.324
C09727=1235.576,159.080,-51.994,-177.746,5.678,148.324
C09728=1235.581,158.830,-51.973,-177.749,5.676,148.325
C09729=1235.586,158.582,-51.951,-177.751,5.675,148.325
C09730=1235.590,158.332,-51.929,-177.754,5.674,148.326
C09731=1235.595,158.084,-51.908,-177.756,5.673,148.326
C09732=1235.600,157.835,-51.886,-177.759,5.671,148.326
C09733=1235.604,157.585,-51.865,-177.761,5.670,148.327
C09734=1235.609,157.337,-51.843,-177.763,5.669,148.327
C09735=1235.614,157.088,-51.821,-177.767,5.668,148.328
C09736=1235.618,156.839,-51.799,-177.769,5.667,148.328
C09737=1235.623,156.589,-51.778,-177.772,5.665,148.329
C09738=1235.628,156.341,-51.756,-177.774,5.664,148.329
C09739=1235.633,156.091,-51.734,-177.776,5.663,148.330
C09740=1235.638,155.842,-51.713,-177.779,5.662,148.330
C09741=1235.642,155.594,-51.692,-177.781,5.661,148.331
C09742=1235.646,155.344,-51.670,-177.784,5.659,148.331
C09743=1235.651,155.095,-51.649,-177.786,5.658,148.332
C09744=1235.656,154.847,-51.628,-177.790,5.657,148.332
C09745=1235.660,154.597,-51.606,-177.792,5.656,148.333
C09746=1235.666,154.348,-51.585,-177.794,5.655,148.333
C09747=1235.671,154.099,-51.563,-177.797,5.653,148.334
C09748=1235.675,153.851,-51.541,-177.799,5.652,148.334
C09749=1235.679,153.601,-51.521,-177.802,5.651,148.335
C09750=1235.684,153.352,-51.499,-177.804,5.650,148.335
C09751=1235.689,153.103,-51.478,-177.807,5.649,148.336
C09752=1235.694,152.854,-51.456,-177.810,5.647,148.336
C09753=1235.698,152.605,-51.434,-177.812,5.646,148.337
C09754=1235.704,152.356,-51.413,-177.815,5.645,148.337
C09755=1235.708,152.108,-51.392,-177.817,5.644,148.338
C09756=1235.712,151.858,-51.371,-177.820,5.643,148.338
C09757=1235.717,151.609,-51.349,-177.823,5.641,148.339
C09758=1235.722,151.360,-51.328,-177.825,5.640,148.339
C09759=1235.727,151.111,-51.306,-177.827,5.639,148.339
C09760=1235.731,150.861,-51.286,-177.830,5.638,148.340
C09761=1235.736,150.613,-51.264,-177.832,5.637,148.340
C09762=1235.741,150.363,-51.243,-177.835,5.635,148.341
C09763=1235.746,150.115,-51.221,-177.837,5.634,148.341
C09764=1235.750,149.865,-51.201,-177.840,5.634,148.342
C09765=1235.755,149.617,-51.179,-177.843,5.632,148.342
C09766=1235.760,149.367,-51.158,-177.845,5.631,148.343
C09767=1235.764,149.119,-51.137,-177.847,5.630,148.343
C09768=1235.769,148.869,-51.116,-177.851,5.629,148.344
C09769=1235.773,148.620,-51.094,-177.853,5.628,148.344
C09770=1235.779,148.371,-51.073,-177.856,5.626,148.345
C09771=1235.783,148.122,-51.053,-177.858,5.625,148.345
C09772=1235.788,147.874,-51.031,-177.860,5.625,148.346
C09773=1235.792,147.624,-51.010,-177.863,5.623,148.346
C09774=1235.797,147.375,-50.989,-177.866,5.622,148.347
C09775=1235.802,147.126,-50.968,-177.868,5.621,148.348
C09776=1235.807,146.877,-50.947,-177.871,5.620,148.348
C09777=1235.811,146.628,-50.925,-177.873,5.619,148.349
C09778=1235.816,146.379,-50.904,-177.875,5.618,148.349
C09779=1235.821,146.129,-50.883,-177.878,5.616,148.350
C09780=1235.825,145.881,-50.862,-177.880,5.615,148.350
C09781=1235.830,145.632,-50.841,-177.884,5.614,148.351
C09782=1235.835,145.382,-50.820,-177.886,5.613,148.351
C09783=1235.840,145.133,-50.800,-177.888,5.612,148.352
C09784=1235.845,144.885,-50.778,-177.891,5.610,148.352
C09785=1235.848,144.635,-50.757,-177.894,5.610,148.353
C09786=1235.854,144.386,-50.736,-177.896,5.609,148.353
C09787=1235.858,144.137,-50.715,-177.899,5.607,148.354
C09788=1235.863,143.888,-50.694,-177.901,5.606,148.354
C09789=1235.868,143.639,-50.673,-177.904,5.605,148.355
C09790=1235.873,143.390,-50.653,-177.906,5.604,148.355
C09791=1235.878,143.141,-50.632,-177.909,5.603,148.356
C09792=1235.881,142.892,-50.611,-177.911,5.602,148.356
C09793=1235.886,142.642,-50.590,-177.914,5.600,148.357
C09794=1235.892,142.393,-50.569,-177.917,5.600,148.357
C09795=1235.896,142.144,-50.548,-177.919,5.599,148.358
C09796=1235.901,141.895,-50.527,-177.922,5.597,148.358
C09797=1235.905,141.647,-50.506,-177.924,5.596,148.359
C09798=1235.911,141.397,-50.485,-177.927,5.596,148.359
C09799=1235.915,141.148,-50.465,-177.929,5.594,148.360
C09800=1235.920,140.899,-50.444,-177.932,5.593,148.360
C09801=1235.925,140.650,-50.424,-177.934,5.592,148.361
C09802=1235.929,140.400,-50.402,-177.937,5.591,148.361
C09803=1235.934,140.151,-50.382,-177.939,5.590,148.362
C09804=1235.939,139.902,-50.361,-177.942,5.589,148.362
C09805=1235.943,139.653,-50.340,-177.944,5.588,148.363
C09806=1235.948,139.405,-50.319,-177.947,5.587,148.363
C09807=1235.952,139.156,-50.298,-177.949,5.586,148.364
C09808=1235.958,138.906,-50.277,-177.952,5.585,148.364
C09809=1235.962,138.657,-50.257,-177.954,5.583,148.365
C09810=1235.967,138.408,-50.236,-177.957,5.583,148.365
C09811=1235.972,138.159,-50.216,-177.959,5.582,148.366
C09812=1235.976,137.910,-50.195,-177.962,5.580,148.366
C09813=1235.981,137.661,-50.174,-177.964,5.579,148.367
C09814=1235.986,137.412,-50.154,-177.967,5.578,148.367
C09815=1235.991,137.163,-50.133,-177.970,5.577,148.368
C09816=1235.995,136.914,-50.113,-177.972,5.576,148.368
C09817=1236.000,136.665,-50.092,-177.975,5.575,148.369
C09818=1236.005,136.416,-50.071,-177.977,5.574,148.369
C09819=1236.009,136.167,-50.051,-177.980,5.573,148.370
C09820=1236.015,135.917,-50.030,-177.982,5.572,148.370
C09821=1236.019,135.668,-50.010,-177.985,5.571,148.371
C09822=1236.024,135.419,-49.990,-177.988,5.569,148.371
C09823=1236.029,135.170,-49.969,-177.990,5.569,148.372
C09824=1236.033,134.921,-49.949,-177.992,5.568,148.372
C09825=1236.039,134.671,-49.928,-177.995,5.566,148.373
C09826=1236.043,134.422,-49.907,-177.998,5.566,148.374
C09827=1236.048,134.154,-49.885,-178.000,5.565,148.374
C09828=1236.053,133.885,-49.863,-178.003,5.563,148.375
C09829=1236.058,133.616,-49.841,-178.006,5.562,148.375
C09830=1236.064,133.347,-49.819,-178.009,5.561,148.376
C09831=1236.068,133.098,-49.799,-178.011,5.560,148.376
C09832=1236.073,132.850,-49.779,-178.014,5.559,148.377
C09833=1236.078,132.600,-49.758,-178.016,5.558,148.377
C09834=1236.082,132.351,-49.737,-178.019,5.557,148.378
C09835=1236.087,132.102,-49.717,-178.021,5.556,148.378
C09836=1236.092,131.852,-49.697,-178.024,5.555,148.379
C09837=1236.097,131.604,-49.676,-178.027,5.554,148.380
C09838=1236.101,131.355,-49.656,-178.029,5.553,148.380
C09839=1236.105,131.106,-49.636,-178.032,5.552,148.381
C09840=1236.111,130.856,-49.615,-178.034,5.551,148.381
C09841=1236.115,130.607,-49.595,-178.037,5.550,148.382
C09842=1236.120,130.358,-49.575,-178.039,5.549,148.382
C09843=1236.125,130.110,-49.555,-178.042,5.548,148.383
C09844=1236.130,129.860,-49.534,-178.044,5.547,148.383
C09845=1236.135,129.611,-49.514,-178.047,5.546,148.384
C09846=1236.139,129.362,-49.494,-178.050,5.545,148.384
C09847=1236.144,129.112,-49.474,-178.052,5.544,148.385
C09848=1236.149,128.863,-49.453,-178.054,5.543,148.385
C09849=1236.153,128.614,-49.433,-178.057,5.542,148.386
C09850=1236.158,128.364,-49.413,-178.060,5.541,148.386
C09851=1236.163,128.116,-49.393,-178.062,5.540,148.387
C09852=1236.167,127.867,-49.372,-178.064,5.539,148.388
C09853=1236.172,127.618,-49.353,-178.067,5.538,148.388
C09854=1236.178,127.368,-49.332,-178.070,5.537,148.389
C09855=1236.182,127.120,-49.312,-178.072,5.536,148.389
C09856=1236.187,126.870,-49.292,-178.075,5.535,148.390
C09857=1236.191,126.621,-49.272,-178.077,5.534,148.390
C09858=1236.196,126.371,-49.252,-178.080,5.533,148.391
C09859=1236.200,126.122,-49.231,-178.082,5.532,148.391
C09860=1236.206,125.874,-49.211,-178.085,5.531,148.392
C09861=1236.211,125.624,-49.191,-178.088,5.530,148.392
C09862=1236.215,125.375,-49.171,-178.090,5.529,148.393
C09863=1236.220,125.126,-49.151,-178.093,5.528,148.394
C09864=1236.225,124.877,-49.131,-178.095,5.527,148.394
C09865=1236.229,124.627,-49.111,-178.098,5.526,148.395
C09866=1236.234,124.379,-49.091,-178.101,5.525,148.395
C09867=1236.239,124.130,-49.072,-178.103,5.524,148.396
C09868=1236.244,123.881,-49.051,-178.105,5.524,148.396
C09869=1236.248,123.631,-49.031,-178.108,5.523,148.397
C09870=1236.253,123.382,-49.011,-178.111,5.521,148.397
C09871=1236.259,123.133,-48.991,-178.113,5.521,148.398
C09872=1236.263,122.884,-48.971,-178.115,5.520,148.398
C09873=1236.268,122.634,-48.951,-178.118,5.519,148.399
C09874=1236.272,122.385,-48.931,-178.121,5.517,148.400
C09875=1236.277,122.136,-48.911,-178.123,5.516,148.400
C09876=1236.282,121.888,-48.891,-178.126,5.516,148.401
C09877=1236.287,121.638,-48.872,-178.128,5.515,148.401
C09878=1236.292,121.388,-48.852,-178.130,5.514,148.402
C09879=1236.296,121.139,-48.831,-178.134,5.513,148.402
C09880=1236.301,120.890,-48.812,-178.136,5.512,148.403
C09881=1236.306,120.642,-48.792,-178.138,5.511,148.403
C09882=1236.311,120.392,-48.772,-178.141,5.510,148.404
C09883=1236.315,120.143,-48.753,-178.143,5.509,148.404
C09884=1236.320,119.894,-48.732,-178.146,5.508,148.405
C09885=1236.325,119.645,-48.713,-178.149,5.507,148.406
C09886=1236.330,119.395,-48.693,-178.151,5.506,148.406
C09887=1236.334,119.146,-48.673,-178.154,5.506,148.407
C09888=1236.340,118.897,-48.654,-178.156,5.505,148.407
C09889=1236.344,118.648,-48.634,-178.159,5.503,148.408
C09890=1236.349,118.399,-48.614,-178.161,5.503,148.408
C09891=1236.353,118.150,-48.594,-178.164,5.502,148.409
C09892=1236.358,117.901,-48.575,-178.166,5.501,148.409
C09893=1236.363,117.651,-48.555,-178.169,5.500,148.410
C09894=1236.367,117.402,-48.535,-178.171,5.499,148.410
C09895=1236.372,117.153,-48.515,-178.174,5.498,148.411
C09896=1236.377,116.904,-48.496,-178.177,5.497,148.412
C09897=1236.382,116.654,-48.477,-178.179,5.496,148.412
C09898=1236.387,116.405,-48.456,-178.181,5.496,148.413
C09899=1236.392,116.156,-48.437,-178.185,5.494,148.413
C09900=1236.397,115.907,-48.417,-178.187,5.493,148.414
C09901=1236.401,115.657,-48.398,-178.189,5.493,148.414
C09902=1236.406,115.409,-48.379,-178.191,5.492,148.415
C09903=1236.411,115.160,-48.358,-178.194,5.491,148.416
C09904=1236.415,114.910,-48.339,-178.197,5.490,148.416
C09905=1236.421,114.661,-48.320,-178.199,5.489,148.417
C09906=1236.425,114.412,-48.300,-178.202,5.488,148.417
C09907=1236.430,114.162,-48.280,-178.205,5.487,148.418
C09908=1236.435,113.913,-48.261,-178.207,5.486,148.418
C09909=1236.439,113.664,-48.242,-178.209,5.486,148.419
C09910=1236.444,113.415,-48.221,-178.212,5.484,148.419
C09911=1236.449,113.166,-48.202,-178.215,5.483,148.420
C09912=1236.454,112.917,-48.183,-178.217,5.483,148.421
C09913=1236.459,112.667,-48.163,-178.220,5.482,148.421
C09914=1236.463,112.419,-48.144,-178.222,5.481,148.422
C09915=1236.468,112.169,-48.125,-178.225,5.480,148.422
C09916=1236.473,111.920,-48.105,-178.228,5.479,148.423
C09917=1236.478,111.671,-48.086,-178.230,5.478,148.423
C09918=1236.483,111.421,-48.066,-178.232,5.477,148.424
C09919=1236.487,111.172,-48.047,-178.235,5.477,148.425
C09920=1236.492,110.923,-48.028,-178.237,5.476,148.425
C09921=1236.498,110.674,-48.008,-178.240,5.475,148.426
C09922=1236.502,110.424,-47.989,-178.242,5.475,148.426
C09923=1236.506,110.175,-47.970,-178.246,5.473,148.427
C09924=1236.512,109.926,-47.950,-178.248,5.472,148.427
C09925=1236.516,109.677,-47.931,-178.250,5.471,148.428
C09926=1236.521,109.428,-47.912,-178.253,5.471,148.429
C09927=1236.526,109.179,-47.892,-178.255,5.470,148.429
C09928=1236.531,108.929,-47.873,-178.258,5.469,148.430
C09929=1236.536,108.680,-47.853,-178.260,5.469,148.430
C09930=1236.540,108.431,-47.834,-178.263,5.467,148.431
C09931=1236.545,108.163,-47.814,-178.266,5.466,148.431
C09932=1236.550,107.894,-47.792,-178.268,5.466,148.432
C09933=1236.556,107.625,-47.772,-178.271,5.464,148.433
C09934=1236.561,107.357,-47.751,-178.274,5.463,148.433
C09935=1236.566,107.107,-47.732,-178.277,5.463,148.434
C09936=1236.570,106.859,-47.713,-178.279,5.462,148.434
C09937=1236.575,106.609,-47.693,-178.281,5.461,148.435
C09938=1236.580,106.361,-47.674,-178.284,5.461,148.436
C09939=1236.584,106.111,-47.655,-178.287,5.459,148.436
C09940=1236.590,105.862,-47.636,-178.289,5.458,148.437
C09941=1236.594,105.613,-47.617,-178.292,5.458,148.437
C09942=1236.599,105.364,-47.598,-178.294,5.457,148.438
C09943=1236.604,105.114,-47.578,-178.297,5.456,148.438
C09944=1236.609,104.866,-47.560,-178.299,5.455,148.439
C09945=1236.614,104.616,-47.540,-178.302,5.455,148.440
C09946=1236.619,104.366,-47.522,-178.304,5.454,148.440
C09947=1236.623,104.117,-47.502,-178.307,5.452,148.441
C09948=1236.629,103.868,-47.483,-178.310,5.452,148.441
C09949=1236.633,103.619,-47.464,-178.312,5.451,148.442
C09950=1236.638,103.370,-47.446,-178.314,5.450,148.442
C09951=1236.642,103.120,-47.426,-178.317,5.449,148.443
C09952=1236.648,102.871,-47.407,-178.320,5.449,148.444
C09953=1236.652,102.622,-47.388,-178.322,5.448,148.444
C09954=1236.657,102.373,-47.370,-178.324,5.447,148.445
C09955=1236.662,102.123,-47.350,-178.327,5.447,148.445
C09956=1236.667,101.875,-47.331,-178.330,5.445,148.446
C09957=1236.671,101.625,-47.312,-178.332,5.444,148.446
C09958=1236.676,101.376,-47.294,-178.335,5.444,148.447
C09959=1236.681,101.126,-47.274,-178.338,5.443,148.448
C09960=1236.686,100.878,-47.255,-178.340,5.442,148.448
C09961=1236.691,100.628,-47.236,-178.342,5.441,148.449
C09962=1236.695,100.379,-47.218,-178.345,5.441,148.449
C09963=1236.700,100.129,-47.198,-178.348,5.440,148.450
C09964=1236.705,99.880,-47.180,-178.350,5.439,148.451
C09965=1236.710,99.631,-47.161,-178.352,5.439,148.451
C09966=1236.715,99.381,-47.142,-178.355,5.437,148.452
C09967=1236.720,99.133,-47.123,-178.358,5.436,148.452
C09968=1236.724,98.883,-47.104,-178.360,5.435,148.453
C09969=1236.730,98.634,-47.085,-178.363,5.435,148.454
C09970=1236.734,98.385,-47.067,-178.365,5.434,148.454
C09971=1236.739,98.135,-47.048,-178.368,5.433,148.455
C09972=1236.744,97.887,-47.029,-178.370,5.433,148.455
C09973=1236.748,97.637,-47.010,-178.373,5.432,148.456
C09974=1236.753,97.388,-46.991,-178.375,5.431,148.457
C09975=1236.758,97.139,-46.973,-178.378,5.430,148.457
C09976=1236.763,96.889,-46.954,-178.380,5.430,148.458
C09977=1236.768,96.641,-46.935,-178.383,5.428,148.458
C09978=1236.772,96.391,-46.917,-178.386,5.428,148.459
C09979=1236.777,96.142,-46.897,-178.388,5.427,148.459
C09980=1236.782,95.893,-46.879,-178.391,5.426,148.460
C09981=1236.787,95.643,-46.860,-178.393,5.426,148.461
C09982=1236.792,95.394,-46.842,-178.396,5.425,148.461
C09983=1236.796,95.145,-46.823,-178.398,5.424,148.462
C09984=1236.802,94.895,-46.804,-178.401,5.423,148.462
C09985=1236.806,94.647,-46.785,-178.403,5.423,148.463
C09986=1236.811,94.397,-46.767,-178.406,5.422,148.464
C09987=1236.816,94.147,-46.749,-178.408,5.421,148.464
C09988=1236.821,93.899,-46.730,-178.411,5.421,148.465
C09989=1236.826,93.648,-46.711,-178.413,5.420,148.465
C09990=1236.830,93.400,-46.692,-178.416,5.419,148.466
C09991=1236.835,93.151,-46.674,-178.419,5.418,148.467
C09992=1236.840,92.901,-46.656,-178.421,5.417,148.467
C09993=1236.845,92.652,-46.637,-178.424,5.416,148.468
C09994=1236.850,92.403,-46.619,-178.426,5.416,148.468
//INST
///DATE 2021/06/25 14:26
///ATTR SC,RW,RJ
////FRAME USER -1
///GROUP1 RB1
NOP
MOVJ C00000 VJ=100.00 PL=0
'Path Start: Op_ID_1
MOVJ C00001 VJ=25.00 PL=0
MOVJ C00002 VJ=25.00 PL=0
'CALL JOB: TOOL ON
MOVL C00003 V=800.0 PL=0
MOVL C00004 V=800.0 PL=0
MOVL C00005 V=800.0 PL=0
MOVL C00006 V=800.0 PL=0
MOVL C00007 V=800.0 PL=0
MOVL C00008 V=800.0 PL=0
MOVL C00009 V=800.0 PL=0
MOVL C00010 V=800.0 PL=0
MOVL C00011 V=800.0 PL=0
MOVL C00012 V=800.0 PL=0
MOVL C00013 V=800.0 PL=0
MOVL C00014 V=800.0 PL=0
MOVL C00015 V=800.0 PL=0
MOVL C00016 V=800.0 PL=0
MOVL C00017 V=800.0 PL=0
MOVL C00018 V=800.0 PL=0
MOVL C00019 V=800.0 PL=0
MOVL C00020 V=800.0 PL=0
MOVL C00021 V=800.0 PL=0
MOVL C00022 V=800.0 PL=0
MOVL C00023 V=800.0 PL=0
MOVL C00024 V=800.0 PL=0
MOVL C00025 V=800.0 PL=0
MOVL C00026 V=800.0 PL=0
MOVL C00027 V=800.0 PL=0
MOVL C00028 V=800.0 PL=0
MOVL C00029 V=800.0 PL=0
MOVL C00030 V=800.0 PL=0
MOVL C00031 V=800.0 PL=0
MOVL C00032 V=800.0 PL=0
MOVL C00033 V=800.0 PL=0
MOVL C00034 V=800.0 PL=0
MOVL C00035 V=800.0 PL=0
MOVL C00036 V=800.0 PL=0
MOVL C00037 V=800.0 PL=0
MOVL C00038 V=800.0 PL=0
MOVL C00039 V=800.0 PL=0
MOVL C00040 V=800.0 PL=0
MOVL C00041 V=800.0 PL=0
MOVL C00042 V=800.0 PL=0
MOVL C00043 V=800.0 PL=0
MOVL C00044 V=800.0 PL=0
MOVL C00045 V=800.0 PL=0
MOVL C00046 V=800.0 PL=0
MOVL C00047 V=800.0 PL=0
MOVL C00048 V=800.0 PL=0
MOVL C00049 V=800.0 PL=0
MOVL C00050 V=800.0 PL=0
MOVL C00051 V=800.0 PL=0
MOVL C00052 V=800.0 PL=0
MOVL C00053 V=800.0 PL=0
MOVL C00054 V=800.0 PL=0
MOVL C00055 V=800.0 PL=0
MOVL C00056 V=800.0 PL=0
MOVL C00057 V=800.0 PL=0
MOVL C00058 V=800.0 PL=0
MOVL C00059 V=800.0 PL=0
MOVL C00060 V=800.0 PL=0
MOVL C00061 V=800.0 PL=0
MOVL C00062 V=800.0 PL=0
MOVL C00063 V=800.0 PL=0
MOVL C00064 V=800.0 PL=0
MOVL C00065 V=800.0 PL=0
MOVL C00066 V=800.0 PL=0
MOVL C00067 V=800.0 PL=0
MOVL C00068 V=800.0 PL=0
MOVL C00069 V=800.0 PL=0
MOVL C00070 V=800.0 PL=0
MOVL C00071 V=800.0 PL=0
MOVL C00072 V=800.0 PL=0
MOVL C00073 V=800.0 PL=0
MOVL C00074 V=800.0 PL=0
MOVL C00075 V=800.0 PL=0
MOVL C00076 V=800.0 PL=0
MOVL C00077 V=800.0 PL=0
MOVL C00078 V=800.0 PL=0
MOVL C00079 V=800.0 PL=0
MOVL C00080 V=800.0 PL=0
MOVL C00081 V=800.0 PL=0
MOVL C00082 V=800.0 PL=0
MOVL C00083 V=800.0 PL=0
MOVL C00084 V=800.0 PL=0
MOVL C00085 V=800.0 PL=0
MOVL C00086 V=800.0 PL=0
MOVL C00087 V=800.0 PL=0
MOVL C00088 V=800.0 PL=0
MOVL C00089 V=800.0 PL=0
MOVL C00090 V=800.0 PL=0
MOVL C00091 V=800.0 PL=0
MOVL C00092 V=800.0 PL=0
MOVL C00093 V=800.0 PL=0
MOVL C00094 V=800.0 PL=0
MOVL C00095 V=800.0 PL=0
MOVL C00096 V=800.0 PL=0
MOVL C00097 V=800.0 PL=0
MOVL C00098 V=800.0 PL=0
MOVL C00099 V=800.0 PL=0
MOVL C00100 V=800.0 PL=0
MOVL C00101 V=800.0 PL=0
MOVL C00102 V=800.0 PL=0
MOVL C00103 V=800.0 PL=0
MOVL C00104 V=800.0 PL=0
MOVL C00105 V=800.0 PL=0
MOVL C00106 V=800.0 PL=0
MOVL C00107 V=800.0 PL=0
MOVL C00108 V=800.0 PL=0
MOVL C00109 V=800.0 PL=0
MOVL C00110 V=800.0 PL=0
MOVL C00111 V=800.0 PL=0
MOVL C00112 V=800.0 PL=0
MOVL C00113 V=800.0 PL=0
MOVL C00114 V=800.0 PL=0
MOVL C00115 V=800.0 PL=0
MOVL C00116 V=800.0 PL=0
MOVL C00117 V=800.0 PL=0
MOVL C00118 V=800.0 PL=0
MOVL C00119 V=800.0 PL=0
MOVL C00120 V=800.0 PL=0
MOVL C00121 V=800.0 PL=0
MOVL C00122 V=800.0 PL=0
MOVL C00123 V=800.0 PL=0
MOVL C00124 V=800.0 PL=0
MOVL C00125 V=800.0 PL=0
MOVL C00126 V=800.0 PL=0
MOVL C00127 V=800.0 PL=0
MOVL C00128 V=800.0 PL=0
MOVL C00129 V=800.0 PL=0
MOVL C00130 V=800.0 PL=0
MOVL C00131 V=800.0 PL=0
MOVL C00132 V=800.0 PL=0
MOVL C00133 V=800.0 PL=0
MOVL C00134 V=800.0 PL=0
MOVL C00135 V=800.0 PL=0
MOVL C00136 V=800.0 PL=0
MOVL C00137 V=800.0 PL=0
MOVL C00138 V=800.0 PL=0
MOVL C00139 V=800.0 PL=0
MOVL C00140 V=800.0 PL=0
MOVL C00141 V=800.0 PL=0
MOVL C00142 V=800.0 PL=0
MOVL C00143 V=800.0 PL=0
MOVL C00144 V=800.0 PL=0
MOVL C00145 V=800.0 PL=0
MOVL C00146 V=800.0 PL=0
MOVL C00147 V=800.0 PL=0
MOVL C00148 V=800.0 PL=0
MOVL C00149 V=800.0 PL=0
MOVL C00150 V=800.0 PL=0
MOVL C00151 V=800.0 PL=0
MOVL C00152 V=800.0 PL=0
MOVL C00153 V=800.0 PL=0
MOVL C00154 V=800.0 PL=0
MOVL C00155 V=800.0 PL=0
MOVL C00156 V=800.0 PL=0
MOVL C00157 V=800.0 PL=0
MOVL C00158 V=800.0 PL=0
MOVL C00159 V=800.0 PL=0
MOVL C00160 V=800.0 PL=0
MOVL C00161 V=800.0 PL=0
MOVL C00162 V=800.0 PL=0
MOVL C00163 V=800.0 PL=0
MOVL C00164 V=800.0 PL=0
MOVL C00165 V=800.0 PL=0
MOVL C00166 V=800.0 PL=0
MOVL C00167 V=800.0 PL=0
MOVL C00168 V=800.0 PL=0
MOVL C00169 V=800.0 PL=0
MOVL C00170 V=800.0 PL=0
MOVL C00171 V=800.0 PL=0
MOVL C00172 V=800.0 PL=0
MOVL C00173 V=800.0 PL=0
MOVL C00174 V=800.0 PL=0
MOVL C00175 V=800.0 PL=0
MOVL C00176 V=800.0 PL=0
MOVL C00177 V=800.0 PL=0
MOVL C00178 V=800.0 PL=0
MOVL C00179 V=800.0 PL=0
MOVL C00180 V=800.0 PL=0
MOVL C00181 V=800.0 PL=0
MOVL C00182 V=800.0 PL=0
MOVL C00183 V=800.0 PL=0
MOVL C00184 V=800.0 PL=0
MOVL C00185 V=800.0 PL=0
MOVL C00186 V=800.0 PL=0
MOVL C00187 V=800.0 PL=0
MOVL C00188 V=800.0 PL=0
MOVL C00189 V=800.0 PL=0
MOVL C00190 V=800.0 PL=0
MOVL C00191 V=800.0 PL=0
MOVL C00192 V=800.0 PL=0
MOVL C00193 V=800.0 PL=0
MOVL C00194 V=800.0 PL=0
MOVL C00195 V=800.0 PL=0
MOVL C00196 V=800.0 PL=0
MOVL C00197 V=800.0 PL=0
MOVL C00198 V=800.0 PL=0
MOVL C00199 V=800.0 PL=0
MOVL C00200 V=800.0 PL=0
MOVL C00201 V=800.0 PL=0
MOVL C00202 V=800.0 PL=0
MOVL C00203 V=800.0 PL=0
MOVL C00204 V=800.0 PL=0
MOVL C00205 V=800.0 PL=0
MOVL C00206 V=800.0 PL=0
MOVL C00207 V=800.0 PL=0
MOVL C00208 V=800.0 PL=0
MOVL C00209 V=800.0 PL=0
MOVL C00210 V=800.0 PL=0
MOVL C00211 V=800.0 PL=0
MOVL C00212 V=800.0 PL=0
MOVL C00213 V=800.0 PL=0
MOVL C00214 V=800.0 PL=0
MOVL C00215 V=800.0 PL=0
MOVL C00216 V=800.0 PL=0
MOVL C00217 V=800.0 PL=0
MOVL C00218 V=800.0 PL=0
MOVL C00219 V=800.0 PL=0
MOVL C00220 V=800.0 PL=0
MOVL C00221 V=800.0 PL=0
MOVL C00222 V=800.0 PL=0
MOVL C00223 V=800.0 PL=0
MOVL C00224 V=800.0 PL=0
MOVL C00225 V=800.0 PL=0
MOVL C00226 V=800.0 PL=0
MOVL C00227 V=800.0 PL=0
MOVL C00228 V=800.0 PL=0
MOVL C00229 V=800.0 PL=0
MOVL C00230 V=800.0 PL=0
MOVL C00231 V=800.0 PL=0
MOVL C00232 V=800.0 PL=0
MOVL C00233 V=800.0 PL=0
MOVL C00234 V=800.0 PL=0
MOVL C00235 V=800.0 PL=0
MOVL C00236 V=800.0 PL=0
MOVL C00237 V=800.0 PL=0
MOVL C00238 V=800.0 PL=0
MOVL C00239 V=800.0 PL=0
MOVL C00240 V=800.0 PL=0
MOVL C00241 V=800.0 PL=0
MOVL C00242 V=800.0 PL=0
MOVL C00243 V=800.0 PL=0
MOVL C00244 V=800.0 PL=0
MOVL C00245 V=800.0 PL=0
MOVL C00246 V=800.0 PL=0
MOVL C00247 V=800.0 PL=0
MOVL C00248 V=800.0 PL=0
MOVL C00249 V=800.0 PL=0
MOVL C00250 V=800.0 PL=0
MOVL C00251 V=800.0 PL=0
MOVL C00252 V=800.0 PL=0
MOVL C00253 V=800.0 PL=0
MOVL C00254 V=800.0 PL=0
MOVL C00255 V=800.0 PL=0
MOVL C00256 V=800.0 PL=0
MOVL C00257 V=800.0 PL=0
MOVL C00258 V=800.0 PL=0
MOVL C00259 V=800.0 PL=0
MOVL C00260 V=800.0 PL=0
MOVL C00261 V=800.0 PL=0
MOVL C00262 V=800.0 PL=0
MOVL C00263 V=800.0 PL=0
MOVL C00264 V=800.0 PL=0
MOVL C00265 V=800.0 PL=0
MOVL C00266 V=800.0 PL=0
MOVL C00267 V=800.0 PL=0
MOVL C00268 V=800.0 PL=0
MOVL C00269 V=800.0 PL=0
MOVL C00270 V=800.0 PL=0
MOVL C00271 V=800.0 PL=0
MOVL C00272 V=800.0 PL=0
MOVL C00273 V=800.0 PL=0
MOVL C00274 V=800.0 PL=0
MOVL C00275 V=800.0 PL=0
MOVL C00276 V=800.0 PL=0
MOVL C00277 V=800.0 PL=0
MOVL C00278 V=800.0 PL=0
MOVL C00279 V=800.0 PL=0
MOVL C00280 V=800.0 PL=0
MOVL C00281 V=800.0 PL=0
MOVL C00282 V=800.0 PL=0
MOVL C00283 V=800.0 PL=0
MOVL C00284 V=800.0 PL=0
MOVL C00285 V=800.0 PL=0
MOVL C00286 V=800.0 PL=0
MOVL C00287 V=800.0 PL=0
MOVL C00288 V=800.0 PL=0
MOVL C00289 V=800.0 PL=0
MOVL C00290 V=800.0 PL=0
MOVL C00291 V=800.0 PL=0
MOVL C00292 V=800.0 PL=0
MOVL C00293 V=800.0 PL=0
MOVL C00294 V=800.0 PL=0
MOVL C00295 V=800.0 PL=0
MOVL C00296 V=800.0 PL=0
MOVL C00297 V=800.0 PL=0
MOVL C00298 V=800.0 PL=0
MOVL C00299 V=800.0 PL=0
MOVL C00300 V=800.0 PL=0
MOVL C00301 V=800.0 PL=0
MOVL C00302 V=800.0 PL=0
MOVL C00303 V=800.0 PL=0
MOVL C00304 V=800.0 PL=0
MOVL C00305 V=800.0 PL=0
MOVL C00306 V=800.0 PL=0
MOVL C00307 V=800.0 PL=0
MOVL C00308 V=800.0 PL=0
MOVL C00309 V=800.0 PL=0
MOVL C00310 V=800.0 PL=0
MOVL C00311 V=800.0 PL=0
MOVL C00312 V=800.0 PL=0
MOVL C00313 V=800.0 PL=0
MOVL C00314 V=800.0 PL=0
MOVL C00315 V=800.0 PL=0
MOVL C00316 V=800.0 PL=0
MOVL C00317 V=800.0 PL=0
MOVL C00318 V=800.0 PL=0
MOVL C00319 V=800.0 PL=0
MOVL C00320 V=800.0 PL=0
MOVL C00321 V=800.0 PL=0
MOVL C00322 V=800.0 PL=0
MOVL C00323 V=800.0 PL=0
MOVL C00324 V=800.0 PL=0
MOVL C00325 V=800.0 PL=0
MOVL C00326 V=800.0 PL=0
MOVL C00327 V=800.0 PL=0
MOVL C00328 V=800.0 PL=0
MOVL C00329 V=800.0 PL=0
MOVL C00330 V=800.0 PL=0
MOVL C00331 V=800.0 PL=0
MOVL C00332 V=800.0 PL=0
MOVL C00333 V=800.0 PL=0
MOVL C00334 V=800.0 PL=0
MOVL C00335 V=800.0 PL=0
MOVL C00336 V=800.0 PL=0
MOVL C00337 V=800.0 PL=0
MOVL C00338 V=800.0 PL=0
MOVL C00339 V=800.0 PL=0
MOVL C00340 V=800.0 PL=0
MOVL C00341 V=800.0 PL=0
MOVL C00342 V=800.0 PL=0
MOVL C00343 V=800.0 PL=0
MOVL C00344 V=800.0 PL=0
MOVL C00345 V=800.0 PL=0
MOVL C00346 V=800.0 PL=0
MOVL C00347 V=800.0 PL=0
MOVL C00348 V=800.0 PL=0
MOVL C00349 V=800.0 PL=0
MOVL C00350 V=800.0 PL=0
MOVL C00351 V=800.0 PL=0
MOVL C00352 V=800.0 PL=0
MOVL C00353 V=800.0 PL=0
MOVL C00354 V=800.0 PL=0
MOVL C00355 V=800.0 PL=0
MOVL C00356 V=800.0 PL=0
MOVL C00357 V=800.0 PL=0
MOVL C00358 V=800.0 PL=0
MOVL C00359 V=800.0 PL=0
MOVL C00360 V=800.0 PL=0
MOVL C00361 V=800.0 PL=0
MOVL C00362 V=800.0 PL=0
MOVL C00363 V=800.0 PL=0
MOVL C00364 V=800.0 PL=0
MOVL C00365 V=800.0 PL=0
MOVL C00366 V=800.0 PL=0
MOVL C00367 V=800.0 PL=0
MOVL C00368 V=800.0 PL=0
MOVL C00369 V=800.0 PL=0
MOVL C00370 V=800.0 PL=0
MOVL C00371 V=800.0 PL=0
MOVL C00372 V=800.0 PL=0
MOVL C00373 V=800.0 PL=0
MOVL C00374 V=800.0 PL=0
MOVL C00375 V=800.0 PL=0
MOVL C00376 V=800.0 PL=0
MOVL C00377 V=800.0 PL=0
MOVL C00378 V=800.0 PL=0
MOVL C00379 V=800.0 PL=0
MOVL C00380 V=800.0 PL=0
MOVL C00381 V=800.0 PL=0
MOVL C00382 V=800.0 PL=0
MOVL C00383 V=800.0 PL=0
MOVL C00384 V=800.0 PL=0
MOVL C00385 V=800.0 PL=0
MOVL C00386 V=800.0 PL=0
MOVL C00387 V=800.0 PL=0
MOVL C00388 V=800.0 PL=0
MOVL C00389 V=800.0 PL=0
MOVL C00390 V=800.0 PL=0
MOVL C00391 V=800.0 PL=0
MOVL C00392 V=800.0 PL=0
MOVL C00393 V=800.0 PL=0
MOVL C00394 V=800.0 PL=0
MOVL C00395 V=800.0 PL=0
MOVL C00396 V=800.0 PL=0
MOVL C00397 V=800.0 PL=0
MOVL C00398 V=800.0 PL=0
MOVL C00399 V=800.0 PL=0
MOVL C00400 V=800.0 PL=0
MOVL C00401 V=800.0 PL=0
MOVL C00402 V=800.0 PL=0
MOVL C00403 V=800.0 PL=0
MOVL C00404 V=800.0 PL=0
MOVL C00405 V=800.0 PL=0
MOVL C00406 V=800.0 PL=0
MOVL C00407 V=800.0 PL=0
MOVL C00408 V=800.0 PL=0
MOVL C00409 V=800.0 PL=0
MOVL C00410 V=800.0 PL=0
MOVL C00411 V=800.0 PL=0
MOVL C00412 V=800.0 PL=0
MOVL C00413 V=800.0 PL=0
MOVL C00414 V=800.0 PL=0
MOVL C00415 V=800.0 PL=0
MOVL C00416 V=800.0 PL=0
MOVL C00417 V=800.0 PL=0
MOVL C00418 V=800.0 PL=0
MOVL C00419 V=800.0 PL=0
MOVL C00420 V=800.0 PL=0
MOVL C00421 V=800.0 PL=0
MOVL C00422 V=800.0 PL=0
MOVL C00423 V=800.0 PL=0
MOVL C00424 V=800.0 PL=0
MOVL C00425 V=800.0 PL=0
MOVL C00426 V=800.0 PL=0
MOVL C00427 V=800.0 PL=0
MOVL C00428 V=800.0 PL=0
MOVL C00429 V=800.0 PL=0
MOVL C00430 V=800.0 PL=0
MOVL C00431 V=800.0 PL=0
MOVL C00432 V=800.0 PL=0
MOVL C00433 V=800.0 PL=0
MOVL C00434 V=800.0 PL=0
MOVL C00435 V=800.0 PL=0
MOVL C00436 V=800.0 PL=0
MOVL C00437 V=800.0 PL=0
MOVL C00438 V=800.0 PL=0
MOVL C00439 V=800.0 PL=0
MOVL C00440 V=800.0 PL=0
MOVL C00441 V=800.0 PL=0
MOVL C00442 V=800.0 PL=0
MOVL C00443 V=800.0 PL=0
MOVL C00444 V=800.0 PL=0
MOVL C00445 V=800.0 PL=0
MOVL C00446 V=800.0 PL=0
MOVL C00447 V=800.0 PL=0
MOVL C00448 V=800.0 PL=0
MOVL C00449 V=800.0 PL=0
MOVL C00450 V=800.0 PL=0
MOVL C00451 V=800.0 PL=0
MOVL C00452 V=800.0 PL=0
MOVL C00453 V=800.0 PL=0
MOVL C00454 V=800.0 PL=0
MOVL C00455 V=800.0 PL=0
MOVL C00456 V=800.0 PL=0
MOVL C00457 V=800.0 PL=0
MOVL C00458 V=800.0 PL=0
MOVL C00459 V=800.0 PL=0
MOVL C00460 V=800.0 PL=0
MOVL C00461 V=800.0 PL=0
MOVL C00462 V=800.0 PL=0
MOVL C00463 V=800.0 PL=0
MOVL C00464 V=800.0 PL=0
MOVL C00465 V=800.0 PL=0
MOVL C00466 V=800.0 PL=0
MOVL C00467 V=800.0 PL=0
MOVL C00468 V=800.0 PL=0
MOVL C00469 V=800.0 PL=0
MOVL C00470 V=800.0 PL=0
MOVL C00471 V=800.0 PL=0
MOVL C00472 V=800.0 PL=0
MOVL C00473 V=800.0 PL=0
MOVL C00474 V=800.0 PL=0
MOVL C00475 V=800.0 PL=0
MOVL C00476 V=800.0 PL=0
MOVL C00477 V=800.0 PL=0
MOVL C00478 V=800.0 PL=0
MOVL C00479 V=800.0 PL=0
MOVL C00480 V=800.0 PL=0
MOVL C00481 V=800.0 PL=0
MOVL C00482 V=800.0 PL=0
MOVL C00483 V=800.0 PL=0
MOVL C00484 V=800.0 PL=0
MOVL C00485 V=800.0 PL=0
MOVL C00486 V=800.0 PL=0
MOVL C00487 V=800.0 PL=0
MOVL C00488 V=800.0 PL=0
MOVL C00489 V=800.0 PL=0
MOVL C00490 V=800.0 PL=0
MOVL C00491 V=800.0 PL=0
MOVL C00492 V=800.0 PL=0
MOVL C00493 V=800.0 PL=0
MOVL C00494 V=800.0 PL=0
MOVL C00495 V=800.0 PL=0
MOVL C00496 V=800.0 PL=0
MOVL C00497 V=800.0 PL=0
MOVL C00498 V=800.0 PL=0
MOVL C00499 V=800.0 PL=0
MOVL C00500 V=800.0 PL=0
MOVL C00501 V=800.0 PL=0
MOVL C00502 V=800.0 PL=0
MOVL C00503 V=800.0 PL=0
MOVL C00504 V=800.0 PL=0
MOVL C00505 V=800.0 PL=0
MOVL C00506 V=800.0 PL=0
MOVL C00507 V=800.0 PL=0
MOVL C00508 V=800.0 PL=0
MOVL C00509 V=800.0 PL=0
MOVL C00510 V=800.0 PL=0
MOVL C00511 V=800.0 PL=0
MOVL C00512 V=800.0 PL=0
MOVL C00513 V=800.0 PL=0
MOVL C00514 V=800.0 PL=0
MOVL C00515 V=800.0 PL=0
MOVL C00516 V=800.0 PL=0
MOVL C00517 V=800.0 PL=0
MOVL C00518 V=800.0 PL=0
MOVL C00519 V=800.0 PL=0
MOVL C00520 V=800.0 PL=0
MOVL C00521 V=800.0 PL=0
MOVL C00522 V=800.0 PL=0
MOVL C00523 V=800.0 PL=0
MOVL C00524 V=800.0 PL=0
MOVL C00525 V=800.0 PL=0
MOVL C00526 V=800.0 PL=0
MOVL C00527 V=800.0 PL=0
MOVL C00528 V=800.0 PL=0
MOVL C00529 V=800.0 PL=0
MOVL C00530 V=800.0 PL=0
MOVL C00531 V=800.0 PL=0
MOVL C00532 V=800.0 PL=0
MOVL C00533 V=800.0 PL=0
MOVL C00534 V=800.0 PL=0
MOVL C00535 V=800.0 PL=0
MOVL C00536 V=800.0 PL=0
MOVL C00537 V=800.0 PL=0
MOVL C00538 V=800.0 PL=0
MOVL C00539 V=800.0 PL=0
MOVL C00540 V=800.0 PL=0
MOVL C00541 V=800.0 PL=0
MOVL C00542 V=800.0 PL=0
MOVL C00543 V=800.0 PL=0
MOVL C00544 V=800.0 PL=0
MOVL C00545 V=800.0 PL=0
MOVL C00546 V=800.0 PL=0
MOVL C00547 V=800.0 PL=0
MOVL C00548 V=800.0 PL=0
MOVL C00549 V=800.0 PL=0
MOVL C00550 V=800.0 PL=0
MOVL C00551 V=800.0 PL=0
MOVL C00552 V=800.0 PL=0
MOVL C00553 V=800.0 PL=0
MOVL C00554 V=800.0 PL=0
MOVL C00555 V=800.0 PL=0
MOVL C00556 V=800.0 PL=0
MOVL C00557 V=800.0 PL=0
MOVL C00558 V=800.0 PL=0
MOVL C00559 V=800.0 PL=0
MOVL C00560 V=800.0 PL=0
MOVL C00561 V=800.0 PL=0
MOVL C00562 V=800.0 PL=0
MOVL C00563 V=800.0 PL=0
MOVL C00564 V=800.0 PL=0
MOVL C00565 V=800.0 PL=0
MOVL C00566 V=800.0 PL=0
MOVL C00567 V=800.0 PL=0
MOVL C00568 V=800.0 PL=0
MOVL C00569 V=800.0 PL=0
MOVL C00570 V=800.0 PL=0
MOVL C00571 V=800.0 PL=0
MOVL C00572 V=800.0 PL=0
MOVL C00573 V=800.0 PL=0
MOVL C00574 V=800.0 PL=0
MOVL C00575 V=800.0 PL=0
MOVL C00576 V=800.0 PL=0
MOVL C00577 V=800.0 PL=0
MOVL C00578 V=800.0 PL=0
MOVL C00579 V=800.0 PL=0
MOVL C00580 V=800.0 PL=0
MOVL C00581 V=800.0 PL=0
MOVL C00582 V=800.0 PL=0
MOVL C00583 V=800.0 PL=0
MOVL C00584 V=800.0 PL=0
MOVL C00585 V=800.0 PL=0
MOVL C00586 V=800.0 PL=0
MOVL C00587 V=800.0 PL=0
MOVL C00588 V=800.0 PL=0
MOVL C00589 V=800.0 PL=0
MOVL C00590 V=800.0 PL=0
MOVL C00591 V=800.0 PL=0
MOVL C00592 V=800.0 PL=0
MOVL C00593 V=800.0 PL=0
MOVL C00594 V=800.0 PL=0
MOVL C00595 V=800.0 PL=0
MOVL C00596 V=800.0 PL=0
MOVL C00597 V=800.0 PL=0
MOVL C00598 V=800.0 PL=0
MOVL C00599 V=800.0 PL=0
MOVL C00600 V=800.0 PL=0
MOVL C00601 V=800.0 PL=0
MOVL C00602 V=800.0 PL=0
MOVL C00603 V=800.0 PL=0
MOVL C00604 V=800.0 PL=0
MOVL C00605 V=800.0 PL=0
MOVL C00606 V=800.0 PL=0
MOVL C00607 V=800.0 PL=0
MOVL C00608 V=800.0 PL=0
MOVL C00609 V=800.0 PL=0
MOVL C00610 V=800.0 PL=0
MOVL C00611 V=800.0 PL=0
MOVL C00612 V=800.0 PL=0
MOVL C00613 V=800.0 PL=0
MOVL C00614 V=800.0 PL=0
MOVL C00615 V=800.0 PL=0
MOVL C00616 V=800.0 PL=0
MOVL C00617 V=800.0 PL=0
MOVL C00618 V=800.0 PL=0
MOVL C00619 V=800.0 PL=0
MOVL C00620 V=800.0 PL=0
MOVL C00621 V=800.0 PL=0
MOVL C00622 V=800.0 PL=0
MOVL C00623 V=800.0 PL=0
MOVL C00624 V=800.0 PL=0
MOVL C00625 V=800.0 PL=0
MOVL C00626 V=800.0 PL=0
MOVL C00627 V=800.0 PL=0
MOVL C00628 V=800.0 PL=0
MOVL C00629 V=800.0 PL=0
MOVL C00630 V=800.0 PL=0
MOVL C00631 V=800.0 PL=0
MOVL C00632 V=800.0 PL=0
MOVL C00633 V=800.0 PL=0
MOVL C00634 V=800.0 PL=0
MOVL C00635 V=800.0 PL=0
MOVL C00636 V=800.0 PL=0
MOVL C00637 V=800.0 PL=0
MOVL C00638 V=800.0 PL=0
MOVL C00639 V=800.0 PL=0
MOVL C00640 V=800.0 PL=0
MOVL C00641 V=800.0 PL=0
MOVL C00642 V=800.0 PL=0
MOVL C00643 V=800.0 PL=0
MOVL C00644 V=800.0 PL=0
MOVL C00645 V=800.0 PL=0
MOVL C00646 V=800.0 PL=0
MOVL C00647 V=800.0 PL=0
MOVL C00648 V=800.0 PL=0
MOVL C00649 V=800.0 PL=0
MOVL C00650 V=800.0 PL=0
MOVL C00651 V=800.0 PL=0
MOVL C00652 V=800.0 PL=0
MOVL C00653 V=800.0 PL=0
MOVL C00654 V=800.0 PL=0
MOVL C00655 V=800.0 PL=0
MOVL C00656 V=800.0 PL=0
MOVL C00657 V=800.0 PL=0
MOVL C00658 V=800.0 PL=0
MOVL C00659 V=800.0 PL=0
MOVL C00660 V=800.0 PL=0
MOVL C00661 V=800.0 PL=0
MOVL C00662 V=800.0 PL=0
MOVL C00663 V=800.0 PL=0
MOVL C00664 V=800.0 PL=0
MOVL C00665 V=800.0 PL=0
MOVL C00666 V=800.0 PL=0
MOVL C00667 V=800.0 PL=0
MOVL C00668 V=800.0 PL=0
MOVL C00669 V=800.0 PL=0
MOVL C00670 V=800.0 PL=0
MOVL C00671 V=800.0 PL=0
MOVL C00672 V=800.0 PL=0
MOVL C00673 V=800.0 PL=0
MOVL C00674 V=800.0 PL=0
MOVL C00675 V=800.0 PL=0
MOVL C00676 V=800.0 PL=0
MOVL C00677 V=800.0 PL=0
MOVL C00678 V=800.0 PL=0
MOVL C00679 V=800.0 PL=0
MOVL C00680 V=800.0 PL=0
MOVL C00681 V=800.0 PL=0
MOVL C00682 V=800.0 PL=0
MOVL C00683 V=800.0 PL=0
MOVL C00684 V=800.0 PL=0
MOVL C00685 V=800.0 PL=0
MOVL C00686 V=800.0 PL=0
MOVL C00687 V=800.0 PL=0
MOVL C00688 V=800.0 PL=0
MOVL C00689 V=800.0 PL=0
MOVL C00690 V=800.0 PL=0
MOVL C00691 V=800.0 PL=0
MOVL C00692 V=800.0 PL=0
MOVL C00693 V=800.0 PL=0
MOVL C00694 V=800.0 PL=0
MOVL C00695 V=800.0 PL=0
MOVL C00696 V=800.0 PL=0
MOVL C00697 V=800.0 PL=0
MOVL C00698 V=800.0 PL=0
MOVL C00699 V=800.0 PL=0
MOVL C00700 V=800.0 PL=0
MOVL C00701 V=800.0 PL=0
MOVL C00702 V=800.0 PL=0
MOVL C00703 V=800.0 PL=0
MOVL C00704 V=800.0 PL=0
MOVL C00705 V=800.0 PL=0
MOVL C00706 V=800.0 PL=0
MOVL C00707 V=800.0 PL=0
MOVL C00708 V=800.0 PL=0
MOVL C00709 V=800.0 PL=0
MOVL C00710 V=800.0 PL=0
MOVL C00711 V=800.0 PL=0
MOVL C00712 V=800.0 PL=0
MOVL C00713 V=800.0 PL=0
MOVL C00714 V=800.0 PL=0
MOVL C00715 V=800.0 PL=0
MOVL C00716 V=800.0 PL=0
MOVL C00717 V=800.0 PL=0
MOVL C00718 V=800.0 PL=0
MOVL C00719 V=800.0 PL=0
MOVL C00720 V=800.0 PL=0
MOVL C00721 V=800.0 PL=0
MOVL C00722 V=800.0 PL=0
MOVL C00723 V=800.0 PL=0
MOVL C00724 V=800.0 PL=0
MOVL C00725 V=800.0 PL=0
MOVL C00726 V=800.0 PL=0
MOVL C00727 V=800.0 PL=0
MOVL C00728 V=800.0 PL=0
MOVL C00729 V=800.0 PL=0
MOVL C00730 V=800.0 PL=0
MOVL C00731 V=800.0 PL=0
MOVL C00732 V=800.0 PL=0
MOVL C00733 V=800.0 PL=0
MOVL C00734 V=800.0 PL=0
MOVL C00735 V=800.0 PL=0
MOVL C00736 V=800.0 PL=0
MOVL C00737 V=800.0 PL=0
MOVL C00738 V=800.0 PL=0
MOVL C00739 V=800.0 PL=0
MOVL C00740 V=800.0 PL=0
MOVL C00741 V=800.0 PL=0
MOVL C00742 V=800.0 PL=0
MOVL C00743 V=800.0 PL=0
MOVL C00744 V=800.0 PL=0
MOVL C00745 V=800.0 PL=0
MOVL C00746 V=800.0 PL=0
MOVL C00747 V=800.0 PL=0
MOVL C00748 V=800.0 PL=0
MOVL C00749 V=800.0 PL=0
MOVL C00750 V=800.0 PL=0
MOVL C00751 V=800.0 PL=0
MOVL C00752 V=800.0 PL=0
MOVL C00753 V=800.0 PL=0
MOVL C00754 V=800.0 PL=0
MOVL C00755 V=800.0 PL=0
MOVL C00756 V=800.0 PL=0
MOVL C00757 V=800.0 PL=0
MOVL C00758 V=800.0 PL=0
MOVL C00759 V=800.0 PL=0
MOVL C00760 V=800.0 PL=0
MOVL C00761 V=800.0 PL=0
MOVL C00762 V=800.0 PL=0
MOVL C00763 V=800.0 PL=0
MOVL C00764 V=800.0 PL=0
MOVL C00765 V=800.0 PL=0
MOVL C00766 V=800.0 PL=0
MOVL C00767 V=800.0 PL=0
MOVL C00768 V=800.0 PL=0
MOVL C00769 V=800.0 PL=0
MOVL C00770 V=800.0 PL=0
MOVL C00771 V=800.0 PL=0
MOVL C00772 V=800.0 PL=0
MOVL C00773 V=800.0 PL=0
MOVL C00774 V=800.0 PL=0
MOVL C00775 V=800.0 PL=0
MOVL C00776 V=800.0 PL=0
MOVL C00777 V=800.0 PL=0
MOVL C00778 V=800.0 PL=0
MOVL C00779 V=800.0 PL=0
MOVL C00780 V=800.0 PL=0
MOVL C00781 V=800.0 PL=0
MOVL C00782 V=800.0 PL=0
MOVL C00783 V=800.0 PL=0
MOVL C00784 V=800.0 PL=0
MOVL C00785 V=800.0 PL=0
MOVL C00786 V=800.0 PL=0
MOVL C00787 V=800.0 PL=0
MOVL C00788 V=800.0 PL=0
MOVL C00789 V=800.0 PL=0
MOVL C00790 V=800.0 PL=0
MOVL C00791 V=800.0 PL=0
MOVL C00792 V=800.0 PL=0
MOVL C00793 V=800.0 PL=0
MOVL C00794 V=800.0 PL=0
MOVL C00795 V=800.0 PL=0
MOVL C00796 V=800.0 PL=0
MOVL C00797 V=800.0 PL=0
MOVL C00798 V=800.0 PL=0
MOVL C00799 V=800.0 PL=0
MOVL C00800 V=800.0 PL=0
MOVL C00801 V=800.0 PL=0
MOVL C00802 V=800.0 PL=0
MOVL C00803 V=800.0 PL=0
MOVL C00804 V=800.0 PL=0
MOVL C00805 V=800.0 PL=0
MOVL C00806 V=800.0 PL=0
MOVL C00807 V=800.0 PL=0
MOVL C00808 V=800.0 PL=0
MOVL C00809 V=800.0 PL=0
MOVL C00810 V=800.0 PL=0
MOVL C00811 V=800.0 PL=0
MOVL C00812 V=800.0 PL=0
MOVL C00813 V=800.0 PL=0
MOVL C00814 V=800.0 PL=0
MOVL C00815 V=800.0 PL=0
MOVL C00816 V=800.0 PL=0
MOVL C00817 V=800.0 PL=0
MOVL C00818 V=800.0 PL=0
MOVL C00819 V=800.0 PL=0
MOVL C00820 V=800.0 PL=0
MOVL C00821 V=800.0 PL=0
MOVL C00822 V=800.0 PL=0
MOVL C00823 V=800.0 PL=0
MOVL C00824 V=800.0 PL=0
MOVL C00825 V=800.0 PL=0
MOVL C00826 V=800.0 PL=0
MOVL C00827 V=800.0 PL=0
MOVL C00828 V=800.0 PL=0
MOVL C00829 V=800.0 PL=0
MOVL C00830 V=800.0 PL=0
MOVL C00831 V=800.0 PL=0
MOVL C00832 V=800.0 PL=0
MOVL C00833 V=800.0 PL=0
MOVL C00834 V=800.0 PL=0
MOVL C00835 V=800.0 PL=0
MOVL C00836 V=800.0 PL=0
MOVL C00837 V=800.0 PL=0
MOVL C00838 V=800.0 PL=0
MOVL C00839 V=800.0 PL=0
MOVL C00840 V=800.0 PL=0
MOVL C00841 V=800.0 PL=0
MOVL C00842 V=800.0 PL=0
MOVL C00843 V=800.0 PL=0
MOVL C00844 V=800.0 PL=0
MOVL C00845 V=800.0 PL=0
MOVL C00846 V=800.0 PL=0
MOVL C00847 V=800.0 PL=0
MOVL C00848 V=800.0 PL=0
MOVL C00849 V=800.0 PL=0
MOVL C00850 V=800.0 PL=0
MOVL C00851 V=800.0 PL=0
MOVL C00852 V=800.0 PL=0
MOVL C00853 V=800.0 PL=0
MOVL C00854 V=800.0 PL=0
MOVL C00855 V=800.0 PL=0
MOVL C00856 V=800.0 PL=0
MOVL C00857 V=800.0 PL=0
MOVL C00858 V=800.0 PL=0
MOVL C00859 V=800.0 PL=0
MOVL C00860 V=800.0 PL=0
MOVL C00861 V=800.0 PL=0
MOVL C00862 V=800.0 PL=0
MOVL C00863 V=800.0 PL=0
MOVL C00864 V=800.0 PL=0
MOVL C00865 V=800.0 PL=0
MOVL C00866 V=800.0 PL=0
MOVL C00867 V=800.0 PL=0
MOVL C00868 V=800.0 PL=0
MOVL C00869 V=800.0 PL=0
MOVL C00870 V=800.0 PL=0
MOVL C00871 V=800.0 PL=0
MOVL C00872 V=800.0 PL=0
MOVL C00873 V=800.0 PL=0
MOVL C00874 V=800.0 PL=0
MOVL C00875 V=800.0 PL=0
MOVL C00876 V=800.0 PL=0
MOVL C00877 V=800.0 PL=0
MOVL C00878 V=800.0 PL=0
MOVL C00879 V=800.0 PL=0
MOVL C00880 V=800.0 PL=0
MOVL C00881 V=800.0 PL=0
MOVL C00882 V=800.0 PL=0
MOVL C00883 V=800.0 PL=0
MOVL C00884 V=800.0 PL=0
MOVL C00885 V=800.0 PL=0
MOVL C00886 V=800.0 PL=0
MOVL C00887 V=800.0 PL=0
MOVL C00888 V=800.0 PL=0
MOVL C00889 V=800.0 PL=0
MOVL C00890 V=800.0 PL=0
MOVL C00891 V=800.0 PL=0
MOVL C00892 V=800.0 PL=0
MOVL C00893 V=800.0 PL=0
MOVL C00894 V=800.0 PL=0
MOVL C00895 V=800.0 PL=0
MOVL C00896 V=800.0 PL=0
MOVL C00897 V=800.0 PL=0
MOVL C00898 V=800.0 PL=0
MOVL C00899 V=800.0 PL=0
MOVL C00900 V=800.0 PL=0
MOVL C00901 V=800.0 PL=0
MOVL C00902 V=800.0 PL=0
MOVL C00903 V=800.0 PL=0
MOVL C00904 V=800.0 PL=0
MOVL C00905 V=800.0 PL=0
MOVL C00906 V=800.0 PL=0
MOVL C00907 V=800.0 PL=0
MOVL C00908 V=800.0 PL=0
MOVL C00909 V=800.0 PL=0
MOVL C00910 V=800.0 PL=0
MOVL C00911 V=800.0 PL=0
MOVL C00912 V=800.0 PL=0
MOVL C00913 V=800.0 PL=0
MOVL C00914 V=800.0 PL=0
MOVL C00915 V=800.0 PL=0
MOVL C00916 V=800.0 PL=0
MOVL C00917 V=800.0 PL=0
MOVL C00918 V=800.0 PL=0
MOVL C00919 V=800.0 PL=0
MOVL C00920 V=800.0 PL=0
MOVL C00921 V=800.0 PL=0
MOVL C00922 V=800.0 PL=0
MOVL C00923 V=800.0 PL=0
MOVL C00924 V=800.0 PL=0
MOVL C00925 V=800.0 PL=0
MOVL C00926 V=800.0 PL=0
MOVL C00927 V=800.0 PL=0
MOVL C00928 V=800.0 PL=0
MOVL C00929 V=800.0 PL=0
MOVL C00930 V=800.0 PL=0
MOVL C00931 V=800.0 PL=0
MOVL C00932 V=800.0 PL=0
MOVL C00933 V=800.0 PL=0
MOVL C00934 V=800.0 PL=0
MOVL C00935 V=800.0 PL=0
MOVL C00936 V=800.0 PL=0
MOVL C00937 V=800.0 PL=0
MOVL C00938 V=800.0 PL=0
MOVL C00939 V=800.0 PL=0
MOVL C00940 V=800.0 PL=0
MOVL C00941 V=800.0 PL=0
MOVL C00942 V=800.0 PL=0
MOVL C00943 V=800.0 PL=0
MOVL C00944 V=800.0 PL=0
MOVL C00945 V=800.0 PL=0
MOVL C00946 V=800.0 PL=0
MOVL C00947 V=800.0 PL=0
MOVL C00948 V=800.0 PL=0
MOVL C00949 V=800.0 PL=0
MOVL C00950 V=800.0 PL=0
MOVL C00951 V=800.0 PL=0
MOVL C00952 V=800.0 PL=0
MOVL C00953 V=800.0 PL=0
MOVL C00954 V=800.0 PL=0
MOVL C00955 V=800.0 PL=0
MOVL C00956 V=800.0 PL=0
MOVL C00957 V=800.0 PL=0
MOVL C00958 V=800.0 PL=0
MOVL C00959 V=800.0 PL=0
MOVL C00960 V=800.0 PL=0
MOVL C00961 V=800.0 PL=0
MOVL C00962 V=800.0 PL=0
MOVL C00963 V=800.0 PL=0
MOVL C00964 V=800.0 PL=0
MOVL C00965 V=800.0 PL=0
MOVL C00966 V=800.0 PL=0
MOVL C00967 V=800.0 PL=0
MOVL C00968 V=800.0 PL=0
MOVL C00969 V=800.0 PL=0
MOVL C00970 V=800.0 PL=0
MOVL C00971 V=800.0 PL=0
MOVL C00972 V=800.0 PL=0
MOVL C00973 V=800.0 PL=0
MOVL C00974 V=800.0 PL=0
MOVL C00975 V=800.0 PL=0
MOVL C00976 V=800.0 PL=0
MOVL C00977 V=800.0 PL=0
MOVL C00978 V=800.0 PL=0
MOVL C00979 V=800.0 PL=0
MOVL C00980 V=800.0 PL=0
MOVL C00981 V=800.0 PL=0
MOVL C00982 V=800.0 PL=0
MOVL C00983 V=800.0 PL=0
MOVL C00984 V=800.0 PL=0
MOVL C00985 V=800.0 PL=0
MOVL C00986 V=800.0 PL=0
MOVL C00987 V=800.0 PL=0
MOVL C00988 V=800.0 PL=0
MOVL C00989 V=800.0 PL=0
MOVL C00990 V=800.0 PL=0
MOVL C00991 V=800.0 PL=0
MOVL C00992 V=800.0 PL=0
MOVL C00993 V=800.0 PL=0
MOVL C00994 V=800.0 PL=0
MOVL C00995 V=800.0 PL=0
MOVL C00996 V=800.0 PL=0
MOVL C00997 V=800.0 PL=0
MOVL C00998 V=800.0 PL=0
MOVL C00999 V=800.0 PL=0
MOVL C01000 V=800.0 PL=0
MOVL C01001 V=800.0 PL=0
MOVL C01002 V=800.0 PL=0
MOVL C01003 V=800.0 PL=0
MOVL C01004 V=800.0 PL=0
MOVL C01005 V=800.0 PL=0
MOVL C01006 V=800.0 PL=0
MOVL C01007 V=800.0 PL=0
MOVL C01008 V=800.0 PL=0
MOVL C01009 V=800.0 PL=0
MOVL C01010 V=800.0 PL=0
MOVL C01011 V=800.0 PL=0
MOVL C01012 V=800.0 PL=0
MOVL C01013 V=800.0 PL=0
MOVL C01014 V=800.0 PL=0
MOVL C01015 V=800.0 PL=0
MOVL C01016 V=800.0 PL=0
MOVL C01017 V=800.0 PL=0
MOVL C01018 V=800.0 PL=0
MOVL C01019 V=800.0 PL=0
MOVL C01020 V=800.0 PL=0
MOVL C01021 V=800.0 PL=0
MOVL C01022 V=800.0 PL=0
MOVL C01023 V=800.0 PL=0
MOVL C01024 V=800.0 PL=0
MOVL C01025 V=800.0 PL=0
MOVL C01026 V=800.0 PL=0
MOVL C01027 V=800.0 PL=0
MOVL C01028 V=800.0 PL=0
MOVL C01029 V=800.0 PL=0
MOVL C01030 V=800.0 PL=0
MOVL C01031 V=800.0 PL=0
MOVL C01032 V=800.0 PL=0
MOVL C01033 V=800.0 PL=0
MOVL C01034 V=800.0 PL=0
MOVL C01035 V=800.0 PL=0
MOVL C01036 V=800.0 PL=0
MOVL C01037 V=800.0 PL=0
MOVL C01038 V=800.0 PL=0
MOVL C01039 V=800.0 PL=0
MOVL C01040 V=800.0 PL=0
MOVL C01041 V=800.0 PL=0
MOVL C01042 V=800.0 PL=0
MOVL C01043 V=800.0 PL=0
MOVL C01044 V=800.0 PL=0
MOVL C01045 V=800.0 PL=0
MOVL C01046 V=800.0 PL=0
MOVL C01047 V=800.0 PL=0
MOVL C01048 V=800.0 PL=0
MOVL C01049 V=800.0 PL=0
MOVL C01050 V=800.0 PL=0
MOVL C01051 V=800.0 PL=0
MOVL C01052 V=800.0 PL=0
MOVL C01053 V=800.0 PL=0
MOVL C01054 V=800.0 PL=0
MOVL C01055 V=800.0 PL=0
MOVL C01056 V=800.0 PL=0
MOVL C01057 V=800.0 PL=0
MOVL C01058 V=800.0 PL=0
MOVL C01059 V=800.0 PL=0
MOVL C01060 V=800.0 PL=0
MOVL C01061 V=800.0 PL=0
MOVL C01062 V=800.0 PL=0
MOVL C01063 V=800.0 PL=0
MOVL C01064 V=800.0 PL=0
MOVL C01065 V=800.0 PL=0
MOVL C01066 V=800.0 PL=0
MOVL C01067 V=800.0 PL=0
MOVL C01068 V=800.0 PL=0
MOVL C01069 V=800.0 PL=0
MOVL C01070 V=800.0 PL=0
MOVL C01071 V=800.0 PL=0
MOVL C01072 V=800.0 PL=0
MOVL C01073 V=800.0 PL=0
MOVL C01074 V=800.0 PL=0
MOVL C01075 V=800.0 PL=0
MOVL C01076 V=800.0 PL=0
MOVL C01077 V=800.0 PL=0
MOVL C01078 V=800.0 PL=0
MOVL C01079 V=800.0 PL=0
MOVL C01080 V=800.0 PL=0
MOVL C01081 V=800.0 PL=0
MOVL C01082 V=800.0 PL=0
MOVL C01083 V=800.0 PL=0
MOVL C01084 V=800.0 PL=0
MOVL C01085 V=800.0 PL=0
MOVL C01086 V=800.0 PL=0
MOVL C01087 V=800.0 PL=0
MOVL C01088 V=800.0 PL=0
MOVL C01089 V=800.0 PL=0
MOVL C01090 V=800.0 PL=0
MOVL C01091 V=800.0 PL=0
MOVL C01092 V=800.0 PL=0
MOVL C01093 V=800.0 PL=0
MOVL C01094 V=800.0 PL=0
MOVL C01095 V=800.0 PL=0
MOVL C01096 V=800.0 PL=0
MOVL C01097 V=800.0 PL=0
MOVL C01098 V=800.0 PL=0
MOVL C01099 V=800.0 PL=0
MOVL C01100 V=800.0 PL=0
MOVL C01101 V=800.0 PL=0
MOVL C01102 V=800.0 PL=0
MOVL C01103 V=800.0 PL=0
MOVL C01104 V=800.0 PL=0
MOVL C01105 V=800.0 PL=0
MOVL C01106 V=800.0 PL=0
MOVL C01107 V=800.0 PL=0
MOVL C01108 V=800.0 PL=0
MOVL C01109 V=800.0 PL=0
MOVL C01110 V=800.0 PL=0
MOVL C01111 V=800.0 PL=0
MOVL C01112 V=800.0 PL=0
MOVL C01113 V=800.0 PL=0
MOVL C01114 V=800.0 PL=0
MOVL C01115 V=800.0 PL=0
MOVL C01116 V=800.0 PL=0
MOVL C01117 V=800.0 PL=0
MOVL C01118 V=800.0 PL=0
MOVL C01119 V=800.0 PL=0
MOVL C01120 V=800.0 PL=0
MOVL C01121 V=800.0 PL=0
MOVL C01122 V=800.0 PL=0
MOVL C01123 V=800.0 PL=0
MOVL C01124 V=800.0 PL=0
MOVL C01125 V=800.0 PL=0
MOVL C01126 V=800.0 PL=0
MOVL C01127 V=800.0 PL=0
MOVL C01128 V=800.0 PL=0
MOVL C01129 V=800.0 PL=0
MOVL C01130 V=800.0 PL=0
MOVL C01131 V=800.0 PL=0
MOVL C01132 V=800.0 PL=0
MOVL C01133 V=800.0 PL=0
MOVL C01134 V=800.0 PL=0
MOVL C01135 V=800.0 PL=0
MOVL C01136 V=800.0 PL=0
MOVL C01137 V=800.0 PL=0
MOVL C01138 V=800.0 PL=0
MOVL C01139 V=800.0 PL=0
MOVL C01140 V=800.0 PL=0
MOVL C01141 V=800.0 PL=0
MOVL C01142 V=800.0 PL=0
MOVL C01143 V=800.0 PL=0
MOVL C01144 V=800.0 PL=0
MOVL C01145 V=800.0 PL=0
MOVL C01146 V=800.0 PL=0
MOVL C01147 V=800.0 PL=0
MOVL C01148 V=800.0 PL=0
MOVL C01149 V=800.0 PL=0
MOVL C01150 V=800.0 PL=0
MOVL C01151 V=800.0 PL=0
MOVL C01152 V=800.0 PL=0
MOVL C01153 V=800.0 PL=0
MOVL C01154 V=800.0 PL=0
MOVL C01155 V=800.0 PL=0
MOVL C01156 V=800.0 PL=0
MOVL C01157 V=800.0 PL=0
MOVL C01158 V=800.0 PL=0
MOVL C01159 V=800.0 PL=0
MOVL C01160 V=800.0 PL=0
MOVL C01161 V=800.0 PL=0
MOVL C01162 V=800.0 PL=0
MOVL C01163 V=800.0 PL=0
MOVL C01164 V=800.0 PL=0
MOVL C01165 V=800.0 PL=0
MOVL C01166 V=800.0 PL=0
MOVL C01167 V=800.0 PL=0
MOVL C01168 V=800.0 PL=0
MOVL C01169 V=800.0 PL=0
MOVL C01170 V=800.0 PL=0
MOVL C01171 V=800.0 PL=0
MOVL C01172 V=800.0 PL=0
MOVL C01173 V=800.0 PL=0
MOVL C01174 V=800.0 PL=0
MOVL C01175 V=800.0 PL=0
MOVL C01176 V=800.0 PL=0
MOVL C01177 V=800.0 PL=0
MOVL C01178 V=800.0 PL=0
MOVL C01179 V=800.0 PL=0
MOVL C01180 V=800.0 PL=0
MOVL C01181 V=800.0 PL=0
MOVL C01182 V=800.0 PL=0
MOVL C01183 V=800.0 PL=0
MOVL C01184 V=800.0 PL=0
MOVL C01185 V=800.0 PL=0
MOVL C01186 V=800.0 PL=0
MOVL C01187 V=800.0 PL=0
MOVL C01188 V=800.0 PL=0
MOVL C01189 V=800.0 PL=0
MOVL C01190 V=800.0 PL=0
MOVL C01191 V=800.0 PL=0
MOVL C01192 V=800.0 PL=0
MOVL C01193 V=800.0 PL=0
MOVL C01194 V=800.0 PL=0
MOVL C01195 V=800.0 PL=0
MOVL C01196 V=800.0 PL=0
MOVL C01197 V=800.0 PL=0
MOVL C01198 V=800.0 PL=0
MOVL C01199 V=800.0 PL=0
MOVL C01200 V=800.0 PL=0
MOVL C01201 V=800.0 PL=0
MOVL C01202 V=800.0 PL=0
MOVL C01203 V=800.0 PL=0
MOVL C01204 V=800.0 PL=0
MOVL C01205 V=800.0 PL=0
MOVL C01206 V=800.0 PL=0
MOVL C01207 V=800.0 PL=0
MOVL C01208 V=800.0 PL=0
MOVL C01209 V=800.0 PL=0
MOVL C01210 V=800.0 PL=0
MOVL C01211 V=800.0 PL=0
MOVL C01212 V=800.0 PL=0
MOVL C01213 V=800.0 PL=0
MOVL C01214 V=800.0 PL=0
MOVL C01215 V=800.0 PL=0
MOVL C01216 V=800.0 PL=0
MOVL C01217 V=800.0 PL=0
MOVL C01218 V=800.0 PL=0
MOVL C01219 V=800.0 PL=0
MOVL C01220 V=800.0 PL=0
MOVL C01221 V=800.0 PL=0
MOVL C01222 V=800.0 PL=0
MOVL C01223 V=800.0 PL=0
MOVL C01224 V=800.0 PL=0
MOVL C01225 V=800.0 PL=0
MOVL C01226 V=800.0 PL=0
MOVL C01227 V=800.0 PL=0
MOVL C01228 V=800.0 PL=0
MOVL C01229 V=800.0 PL=0
MOVL C01230 V=800.0 PL=0
MOVL C01231 V=800.0 PL=0
MOVL C01232 V=800.0 PL=0
MOVL C01233 V=800.0 PL=0
MOVL C01234 V=800.0 PL=0
MOVL C01235 V=800.0 PL=0
MOVL C01236 V=800.0 PL=0
MOVL C01237 V=800.0 PL=0
MOVL C01238 V=800.0 PL=0
MOVL C01239 V=800.0 PL=0
MOVL C01240 V=800.0 PL=0
MOVL C01241 V=800.0 PL=0
MOVL C01242 V=800.0 PL=0
MOVL C01243 V=800.0 PL=0
MOVL C01244 V=800.0 PL=0
MOVL C01245 V=800.0 PL=0
MOVL C01246 V=800.0 PL=0
MOVL C01247 V=800.0 PL=0
MOVL C01248 V=800.0 PL=0
MOVL C01249 V=800.0 PL=0
MOVL C01250 V=800.0 PL=0
MOVL C01251 V=800.0 PL=0
MOVL C01252 V=800.0 PL=0
MOVL C01253 V=800.0 PL=0
MOVL C01254 V=800.0 PL=0
MOVL C01255 V=800.0 PL=0
MOVL C01256 V=800.0 PL=0
MOVL C01257 V=800.0 PL=0
MOVL C01258 V=800.0 PL=0
MOVL C01259 V=800.0 PL=0
MOVL C01260 V=800.0 PL=0
MOVL C01261 V=800.0 PL=0
MOVL C01262 V=800.0 PL=0
MOVL C01263 V=800.0 PL=0
MOVL C01264 V=800.0 PL=0
MOVL C01265 V=800.0 PL=0
MOVL C01266 V=800.0 PL=0
MOVL C01267 V=800.0 PL=0
MOVL C01268 V=800.0 PL=0
MOVL C01269 V=800.0 PL=0
MOVL C01270 V=800.0 PL=0
MOVL C01271 V=800.0 PL=0
MOVL C01272 V=800.0 PL=0
MOVL C01273 V=800.0 PL=0
MOVL C01274 V=800.0 PL=0
MOVL C01275 V=800.0 PL=0
MOVL C01276 V=800.0 PL=0
MOVL C01277 V=800.0 PL=0
MOVL C01278 V=800.0 PL=0
MOVL C01279 V=800.0 PL=0
MOVL C01280 V=800.0 PL=0
MOVL C01281 V=800.0 PL=0
MOVL C01282 V=800.0 PL=0
MOVL C01283 V=800.0 PL=0
MOVL C01284 V=800.0 PL=0
MOVL C01285 V=800.0 PL=0
MOVL C01286 V=800.0 PL=0
MOVL C01287 V=800.0 PL=0
MOVL C01288 V=800.0 PL=0
MOVL C01289 V=800.0 PL=0
MOVL C01290 V=800.0 PL=0
MOVL C01291 V=800.0 PL=0
MOVL C01292 V=800.0 PL=0
MOVL C01293 V=800.0 PL=0
MOVL C01294 V=800.0 PL=0
MOVL C01295 V=800.0 PL=0
MOVL C01296 V=800.0 PL=0
MOVL C01297 V=800.0 PL=0
MOVL C01298 V=800.0 PL=0
MOVL C01299 V=800.0 PL=0
MOVL C01300 V=800.0 PL=0
MOVL C01301 V=800.0 PL=0
MOVL C01302 V=800.0 PL=0
MOVL C01303 V=800.0 PL=0
MOVL C01304 V=800.0 PL=0
MOVL C01305 V=800.0 PL=0
MOVL C01306 V=800.0 PL=0
MOVL C01307 V=800.0 PL=0
MOVL C01308 V=800.0 PL=0
MOVL C01309 V=800.0 PL=0
MOVL C01310 V=800.0 PL=0
MOVL C01311 V=800.0 PL=0
MOVL C01312 V=800.0 PL=0
MOVL C01313 V=800.0 PL=0
MOVL C01314 V=800.0 PL=0
MOVL C01315 V=800.0 PL=0
MOVL C01316 V=800.0 PL=0
MOVL C01317 V=800.0 PL=0
MOVL C01318 V=800.0 PL=0
MOVL C01319 V=800.0 PL=0
MOVL C01320 V=800.0 PL=0
MOVL C01321 V=800.0 PL=0
MOVL C01322 V=800.0 PL=0
MOVL C01323 V=800.0 PL=0
MOVL C01324 V=800.0 PL=0
MOVL C01325 V=800.0 PL=0
MOVL C01326 V=800.0 PL=0
MOVL C01327 V=800.0 PL=0
MOVL C01328 V=800.0 PL=0
MOVL C01329 V=800.0 PL=0
MOVL C01330 V=800.0 PL=0
MOVL C01331 V=800.0 PL=0
MOVL C01332 V=800.0 PL=0
MOVL C01333 V=800.0 PL=0
MOVL C01334 V=800.0 PL=0
MOVL C01335 V=800.0 PL=0
MOVL C01336 V=800.0 PL=0
MOVL C01337 V=800.0 PL=0
MOVL C01338 V=800.0 PL=0
MOVL C01339 V=800.0 PL=0
MOVL C01340 V=800.0 PL=0
MOVL C01341 V=800.0 PL=0
MOVL C01342 V=800.0 PL=0
MOVL C01343 V=800.0 PL=0
MOVL C01344 V=800.0 PL=0
MOVL C01345 V=800.0 PL=0
MOVL C01346 V=800.0 PL=0
MOVL C01347 V=800.0 PL=0
MOVL C01348 V=800.0 PL=0
MOVL C01349 V=800.0 PL=0
MOVL C01350 V=800.0 PL=0
MOVL C01351 V=800.0 PL=0
MOVL C01352 V=800.0 PL=0
MOVL C01353 V=800.0 PL=0
MOVL C01354 V=800.0 PL=0
MOVL C01355 V=800.0 PL=0
MOVL C01356 V=800.0 PL=0
MOVL C01357 V=800.0 PL=0
MOVL C01358 V=800.0 PL=0
MOVL C01359 V=800.0 PL=0
MOVL C01360 V=800.0 PL=0
MOVL C01361 V=800.0 PL=0
MOVL C01362 V=800.0 PL=0
MOVL C01363 V=800.0 PL=0
MOVL C01364 V=800.0 PL=0
MOVL C01365 V=800.0 PL=0
MOVL C01366 V=800.0 PL=0
MOVL C01367 V=800.0 PL=0
MOVL C01368 V=800.0 PL=0
MOVL C01369 V=800.0 PL=0
MOVL C01370 V=800.0 PL=0
MOVL C01371 V=800.0 PL=0
MOVL C01372 V=800.0 PL=0
MOVL C01373 V=800.0 PL=0
MOVL C01374 V=800.0 PL=0
MOVL C01375 V=800.0 PL=0
MOVL C01376 V=800.0 PL=0
MOVL C01377 V=800.0 PL=0
MOVL C01378 V=800.0 PL=0
MOVL C01379 V=800.0 PL=0
MOVL C01380 V=800.0 PL=0
MOVL C01381 V=800.0 PL=0
MOVL C01382 V=800.0 PL=0
MOVL C01383 V=800.0 PL=0
MOVL C01384 V=800.0 PL=0
MOVL C01385 V=800.0 PL=0
MOVL C01386 V=800.0 PL=0
MOVL C01387 V=800.0 PL=0
MOVL C01388 V=800.0 PL=0
MOVL C01389 V=800.0 PL=0
MOVL C01390 V=800.0 PL=0
MOVL C01391 V=800.0 PL=0
MOVL C01392 V=800.0 PL=0
MOVL C01393 V=800.0 PL=0
MOVL C01394 V=800.0 PL=0
MOVL C01395 V=800.0 PL=0
MOVL C01396 V=800.0 PL=0
MOVL C01397 V=800.0 PL=0
MOVL C01398 V=800.0 PL=0
MOVL C01399 V=800.0 PL=0
MOVL C01400 V=800.0 PL=0
MOVL C01401 V=800.0 PL=0
MOVL C01402 V=800.0 PL=0
MOVL C01403 V=800.0 PL=0
MOVL C01404 V=800.0 PL=0
MOVL C01405 V=800.0 PL=0
MOVL C01406 V=800.0 PL=0
MOVL C01407 V=800.0 PL=0
MOVL C01408 V=800.0 PL=0
MOVL C01409 V=800.0 PL=0
MOVL C01410 V=800.0 PL=0
MOVL C01411 V=800.0 PL=0
MOVL C01412 V=800.0 PL=0
MOVL C01413 V=800.0 PL=0
MOVL C01414 V=800.0 PL=0
MOVL C01415 V=800.0 PL=0
MOVL C01416 V=800.0 PL=0
MOVL C01417 V=800.0 PL=0
MOVL C01418 V=800.0 PL=0
MOVL C01419 V=800.0 PL=0
MOVL C01420 V=800.0 PL=0
MOVL C01421 V=800.0 PL=0
MOVL C01422 V=800.0 PL=0
MOVL C01423 V=800.0 PL=0
MOVL C01424 V=800.0 PL=0
MOVL C01425 V=800.0 PL=0
MOVL C01426 V=800.0 PL=0
MOVL C01427 V=800.0 PL=0
MOVL C01428 V=800.0 PL=0
MOVL C01429 V=800.0 PL=0
MOVL C01430 V=800.0 PL=0
MOVL C01431 V=800.0 PL=0
MOVL C01432 V=800.0 PL=0
MOVL C01433 V=800.0 PL=0
MOVL C01434 V=800.0 PL=0
MOVL C01435 V=800.0 PL=0
MOVL C01436 V=800.0 PL=0
MOVL C01437 V=800.0 PL=0
MOVL C01438 V=800.0 PL=0
MOVL C01439 V=800.0 PL=0
MOVL C01440 V=800.0 PL=0
MOVL C01441 V=800.0 PL=0
MOVL C01442 V=800.0 PL=0
MOVL C01443 V=800.0 PL=0
MOVL C01444 V=800.0 PL=0
MOVL C01445 V=800.0 PL=0
MOVL C01446 V=800.0 PL=0
MOVL C01447 V=800.0 PL=0
MOVL C01448 V=800.0 PL=0
MOVL C01449 V=800.0 PL=0
MOVL C01450 V=800.0 PL=0
MOVL C01451 V=800.0 PL=0
MOVL C01452 V=800.0 PL=0
MOVL C01453 V=800.0 PL=0
MOVL C01454 V=800.0 PL=0
MOVL C01455 V=800.0 PL=0
MOVL C01456 V=800.0 PL=0
MOVL C01457 V=800.0 PL=0
MOVL C01458 V=800.0 PL=0
MOVL C01459 V=800.0 PL=0
MOVL C01460 V=800.0 PL=0
MOVL C01461 V=800.0 PL=0
MOVL C01462 V=800.0 PL=0
MOVL C01463 V=800.0 PL=0
MOVL C01464 V=800.0 PL=0
MOVL C01465 V=800.0 PL=0
MOVL C01466 V=800.0 PL=0
MOVL C01467 V=800.0 PL=0
MOVL C01468 V=800.0 PL=0
MOVL C01469 V=800.0 PL=0
MOVL C01470 V=800.0 PL=0
MOVL C01471 V=800.0 PL=0
MOVL C01472 V=800.0 PL=0
MOVL C01473 V=800.0 PL=0
MOVL C01474 V=800.0 PL=0
MOVL C01475 V=800.0 PL=0
MOVL C01476 V=800.0 PL=0
MOVL C01477 V=800.0 PL=0
MOVL C01478 V=800.0 PL=0
MOVL C01479 V=800.0 PL=0
MOVL C01480 V=800.0 PL=0
MOVL C01481 V=800.0 PL=0
MOVL C01482 V=800.0 PL=0
MOVL C01483 V=800.0 PL=0
MOVL C01484 V=800.0 PL=0
MOVL C01485 V=800.0 PL=0
MOVL C01486 V=800.0 PL=0
MOVL C01487 V=800.0 PL=0
MOVL C01488 V=800.0 PL=0
MOVL C01489 V=800.0 PL=0
MOVL C01490 V=800.0 PL=0
MOVL C01491 V=800.0 PL=0
MOVL C01492 V=800.0 PL=0
MOVL C01493 V=800.0 PL=0
MOVL C01494 V=800.0 PL=0
MOVL C01495 V=800.0 PL=0
MOVL C01496 V=800.0 PL=0
MOVL C01497 V=800.0 PL=0
MOVL C01498 V=800.0 PL=0
MOVL C01499 V=800.0 PL=0
MOVL C01500 V=800.0 PL=0
MOVL C01501 V=800.0 PL=0
MOVL C01502 V=800.0 PL=0
MOVL C01503 V=800.0 PL=0
MOVL C01504 V=800.0 PL=0
MOVL C01505 V=800.0 PL=0
MOVL C01506 V=800.0 PL=0
MOVL C01507 V=800.0 PL=0
MOVL C01508 V=800.0 PL=0
MOVL C01509 V=800.0 PL=0
MOVL C01510 V=800.0 PL=0
MOVL C01511 V=800.0 PL=0
MOVL C01512 V=800.0 PL=0
MOVL C01513 V=800.0 PL=0
MOVL C01514 V=800.0 PL=0
MOVL C01515 V=800.0 PL=0
MOVL C01516 V=800.0 PL=0
MOVL C01517 V=800.0 PL=0
MOVL C01518 V=800.0 PL=0
MOVL C01519 V=800.0 PL=0
MOVL C01520 V=800.0 PL=0
MOVL C01521 V=800.0 PL=0
MOVL C01522 V=800.0 PL=0
MOVL C01523 V=800.0 PL=0
MOVL C01524 V=800.0 PL=0
MOVL C01525 V=800.0 PL=0
MOVL C01526 V=800.0 PL=0
MOVL C01527 V=800.0 PL=0
MOVL C01528 V=800.0 PL=0
MOVL C01529 V=800.0 PL=0
MOVL C01530 V=800.0 PL=0
MOVL C01531 V=800.0 PL=0
MOVL C01532 V=800.0 PL=0
MOVL C01533 V=800.0 PL=0
MOVL C01534 V=800.0 PL=0
MOVL C01535 V=800.0 PL=0
MOVL C01536 V=800.0 PL=0
MOVL C01537 V=800.0 PL=0
MOVL C01538 V=800.0 PL=0
MOVL C01539 V=800.0 PL=0
MOVL C01540 V=800.0 PL=0
MOVL C01541 V=800.0 PL=0
MOVL C01542 V=800.0 PL=0
MOVL C01543 V=800.0 PL=0
MOVL C01544 V=800.0 PL=0
MOVL C01545 V=800.0 PL=0
MOVL C01546 V=800.0 PL=0
MOVL C01547 V=800.0 PL=0
MOVL C01548 V=800.0 PL=0
MOVL C01549 V=800.0 PL=0
MOVL C01550 V=800.0 PL=0
MOVL C01551 V=800.0 PL=0
MOVL C01552 V=800.0 PL=0
MOVL C01553 V=800.0 PL=0
MOVL C01554 V=800.0 PL=0
MOVL C01555 V=800.0 PL=0
MOVL C01556 V=800.0 PL=0
MOVL C01557 V=800.0 PL=0
MOVL C01558 V=800.0 PL=0
MOVL C01559 V=800.0 PL=0
MOVL C01560 V=800.0 PL=0
MOVL C01561 V=800.0 PL=0
MOVL C01562 V=800.0 PL=0
MOVL C01563 V=800.0 PL=0
MOVL C01564 V=800.0 PL=0
MOVL C01565 V=800.0 PL=0
MOVL C01566 V=800.0 PL=0
MOVL C01567 V=800.0 PL=0
MOVL C01568 V=800.0 PL=0
MOVL C01569 V=800.0 PL=0
MOVL C01570 V=800.0 PL=0
MOVL C01571 V=800.0 PL=0
MOVL C01572 V=800.0 PL=0
MOVL C01573 V=800.0 PL=0
MOVL C01574 V=800.0 PL=0
MOVL C01575 V=800.0 PL=0
MOVL C01576 V=800.0 PL=0
MOVL C01577 V=800.0 PL=0
MOVL C01578 V=800.0 PL=0
MOVL C01579 V=800.0 PL=0
MOVL C01580 V=800.0 PL=0
MOVL C01581 V=800.0 PL=0
MOVL C01582 V=800.0 PL=0
MOVL C01583 V=800.0 PL=0
MOVL C01584 V=800.0 PL=0
MOVL C01585 V=800.0 PL=0
MOVL C01586 V=800.0 PL=0
MOVL C01587 V=800.0 PL=0
MOVL C01588 V=800.0 PL=0
MOVL C01589 V=800.0 PL=0
MOVL C01590 V=800.0 PL=0
MOVL C01591 V=800.0 PL=0
MOVL C01592 V=800.0 PL=0
MOVL C01593 V=800.0 PL=0
MOVL C01594 V=800.0 PL=0
MOVL C01595 V=800.0 PL=0
MOVL C01596 V=800.0 PL=0
MOVL C01597 V=800.0 PL=0
MOVL C01598 V=800.0 PL=0
MOVL C01599 V=800.0 PL=0
MOVL C01600 V=800.0 PL=0
MOVL C01601 V=800.0 PL=0
MOVL C01602 V=800.0 PL=0
MOVL C01603 V=800.0 PL=0
MOVL C01604 V=800.0 PL=0
MOVL C01605 V=800.0 PL=0
MOVL C01606 V=800.0 PL=0
MOVL C01607 V=800.0 PL=0
MOVL C01608 V=800.0 PL=0
MOVL C01609 V=800.0 PL=0
MOVL C01610 V=800.0 PL=0
MOVL C01611 V=800.0 PL=0
MOVL C01612 V=800.0 PL=0
MOVL C01613 V=800.0 PL=0
MOVL C01614 V=800.0 PL=0
MOVL C01615 V=800.0 PL=0
MOVL C01616 V=800.0 PL=0
MOVL C01617 V=800.0 PL=0
MOVL C01618 V=800.0 PL=0
MOVL C01619 V=800.0 PL=0
MOVL C01620 V=800.0 PL=0
MOVL C01621 V=800.0 PL=0
MOVL C01622 V=800.0 PL=0
MOVL C01623 V=800.0 PL=0
MOVL C01624 V=800.0 PL=0
MOVL C01625 V=800.0 PL=0
MOVL C01626 V=800.0 PL=0
MOVL C01627 V=800.0 PL=0
MOVL C01628 V=800.0 PL=0
MOVL C01629 V=800.0 PL=0
MOVL C01630 V=800.0 PL=0
MOVL C01631 V=800.0 PL=0
MOVL C01632 V=800.0 PL=0
MOVL C01633 V=800.0 PL=0
MOVL C01634 V=800.0 PL=0
MOVL C01635 V=800.0 PL=0
MOVL C01636 V=800.0 PL=0
MOVL C01637 V=800.0 PL=0
MOVL C01638 V=800.0 PL=0
MOVL C01639 V=800.0 PL=0
MOVL C01640 V=800.0 PL=0
MOVL C01641 V=800.0 PL=0
MOVL C01642 V=800.0 PL=0
MOVL C01643 V=800.0 PL=0
MOVL C01644 V=800.0 PL=0
MOVL C01645 V=800.0 PL=0
MOVL C01646 V=800.0 PL=0
MOVL C01647 V=800.0 PL=0
MOVL C01648 V=800.0 PL=0
MOVL C01649 V=800.0 PL=0
MOVL C01650 V=800.0 PL=0
MOVL C01651 V=800.0 PL=0
MOVL C01652 V=800.0 PL=0
MOVL C01653 V=800.0 PL=0
MOVL C01654 V=800.0 PL=0
MOVL C01655 V=800.0 PL=0
MOVL C01656 V=800.0 PL=0
MOVL C01657 V=800.0 PL=0
MOVL C01658 V=800.0 PL=0
MOVL C01659 V=800.0 PL=0
MOVL C01660 V=800.0 PL=0
MOVL C01661 V=800.0 PL=0
MOVL C01662 V=800.0 PL=0
MOVL C01663 V=800.0 PL=0
MOVL C01664 V=800.0 PL=0
MOVL C01665 V=800.0 PL=0
MOVL C01666 V=800.0 PL=0
MOVL C01667 V=800.0 PL=0
MOVL C01668 V=800.0 PL=0
MOVL C01669 V=800.0 PL=0
MOVL C01670 V=800.0 PL=0
MOVL C01671 V=800.0 PL=0
MOVL C01672 V=800.0 PL=0
MOVL C01673 V=800.0 PL=0
MOVL C01674 V=800.0 PL=0
MOVL C01675 V=800.0 PL=0
MOVL C01676 V=800.0 PL=0
MOVL C01677 V=800.0 PL=0
MOVL C01678 V=800.0 PL=0
MOVL C01679 V=800.0 PL=0
MOVL C01680 V=800.0 PL=0
MOVL C01681 V=800.0 PL=0
MOVL C01682 V=800.0 PL=0
MOVL C01683 V=800.0 PL=0
MOVL C01684 V=800.0 PL=0
MOVL C01685 V=800.0 PL=0
MOVL C01686 V=800.0 PL=0
MOVL C01687 V=800.0 PL=0
MOVL C01688 V=800.0 PL=0
MOVL C01689 V=800.0 PL=0
MOVL C01690 V=800.0 PL=0
MOVL C01691 V=800.0 PL=0
MOVL C01692 V=800.0 PL=0
MOVL C01693 V=800.0 PL=0
MOVL C01694 V=800.0 PL=0
MOVL C01695 V=800.0 PL=0
MOVL C01696 V=800.0 PL=0
MOVL C01697 V=800.0 PL=0
MOVL C01698 V=800.0 PL=0
MOVL C01699 V=800.0 PL=0
MOVL C01700 V=800.0 PL=0
MOVL C01701 V=800.0 PL=0
MOVL C01702 V=800.0 PL=0
MOVL C01703 V=800.0 PL=0
MOVL C01704 V=800.0 PL=0
MOVL C01705 V=800.0 PL=0
MOVL C01706 V=800.0 PL=0
MOVL C01707 V=800.0 PL=0
MOVL C01708 V=800.0 PL=0
MOVL C01709 V=800.0 PL=0
MOVL C01710 V=800.0 PL=0
MOVL C01711 V=800.0 PL=0
MOVL C01712 V=800.0 PL=0
MOVL C01713 V=800.0 PL=0
MOVL C01714 V=800.0 PL=0
MOVL C01715 V=800.0 PL=0
MOVL C01716 V=800.0 PL=0
MOVL C01717 V=800.0 PL=0
MOVL C01718 V=800.0 PL=0
MOVL C01719 V=800.0 PL=0
MOVL C01720 V=800.0 PL=0
MOVL C01721 V=800.0 PL=0
MOVL C01722 V=800.0 PL=0
MOVL C01723 V=800.0 PL=0
MOVL C01724 V=800.0 PL=0
MOVL C01725 V=800.0 PL=0
MOVL C01726 V=800.0 PL=0
MOVL C01727 V=800.0 PL=0
MOVL C01728 V=800.0 PL=0
MOVL C01729 V=800.0 PL=0
MOVL C01730 V=800.0 PL=0
MOVL C01731 V=800.0 PL=0
MOVL C01732 V=800.0 PL=0
MOVL C01733 V=800.0 PL=0
MOVL C01734 V=800.0 PL=0
MOVL C01735 V=800.0 PL=0
MOVL C01736 V=800.0 PL=0
MOVL C01737 V=800.0 PL=0
MOVL C01738 V=800.0 PL=0
MOVL C01739 V=800.0 PL=0
MOVL C01740 V=800.0 PL=0
MOVL C01741 V=800.0 PL=0
MOVL C01742 V=800.0 PL=0
MOVL C01743 V=800.0 PL=0
MOVL C01744 V=800.0 PL=0
MOVL C01745 V=800.0 PL=0
MOVL C01746 V=800.0 PL=0
MOVL C01747 V=800.0 PL=0
MOVL C01748 V=800.0 PL=0
MOVL C01749 V=800.0 PL=0
MOVL C01750 V=800.0 PL=0
MOVL C01751 V=800.0 PL=0
MOVL C01752 V=800.0 PL=0
MOVL C01753 V=800.0 PL=0
MOVL C01754 V=800.0 PL=0
MOVL C01755 V=800.0 PL=0
MOVL C01756 V=800.0 PL=0
MOVL C01757 V=800.0 PL=0
MOVL C01758 V=800.0 PL=0
MOVL C01759 V=800.0 PL=0
MOVL C01760 V=800.0 PL=0
MOVL C01761 V=800.0 PL=0
MOVL C01762 V=800.0 PL=0
MOVL C01763 V=800.0 PL=0
MOVL C01764 V=800.0 PL=0
MOVL C01765 V=800.0 PL=0
MOVL C01766 V=800.0 PL=0
MOVL C01767 V=800.0 PL=0
MOVL C01768 V=800.0 PL=0
MOVL C01769 V=800.0 PL=0
MOVL C01770 V=800.0 PL=0
MOVL C01771 V=800.0 PL=0
MOVL C01772 V=800.0 PL=0
MOVL C01773 V=800.0 PL=0
MOVL C01774 V=800.0 PL=0
MOVL C01775 V=800.0 PL=0
MOVL C01776 V=800.0 PL=0
MOVL C01777 V=800.0 PL=0
MOVL C01778 V=800.0 PL=0
MOVL C01779 V=800.0 PL=0
MOVL C01780 V=800.0 PL=0
MOVL C01781 V=800.0 PL=0
MOVL C01782 V=800.0 PL=0
MOVL C01783 V=800.0 PL=0
MOVL C01784 V=800.0 PL=0
MOVL C01785 V=800.0 PL=0
MOVL C01786 V=800.0 PL=0
MOVL C01787 V=800.0 PL=0
MOVL C01788 V=800.0 PL=0
MOVL C01789 V=800.0 PL=0
MOVL C01790 V=800.0 PL=0
MOVL C01791 V=800.0 PL=0
MOVL C01792 V=800.0 PL=0
MOVL C01793 V=800.0 PL=0
MOVL C01794 V=800.0 PL=0
MOVL C01795 V=800.0 PL=0
MOVL C01796 V=800.0 PL=0
MOVL C01797 V=800.0 PL=0
MOVL C01798 V=800.0 PL=0
MOVL C01799 V=800.0 PL=0
MOVL C01800 V=800.0 PL=0
MOVL C01801 V=800.0 PL=0
MOVL C01802 V=800.0 PL=0
MOVL C01803 V=800.0 PL=0
MOVL C01804 V=800.0 PL=0
MOVL C01805 V=800.0 PL=0
MOVL C01806 V=800.0 PL=0
MOVL C01807 V=800.0 PL=0
MOVL C01808 V=800.0 PL=0
MOVL C01809 V=800.0 PL=0
MOVL C01810 V=800.0 PL=0
MOVL C01811 V=800.0 PL=0
MOVL C01812 V=800.0 PL=0
MOVL C01813 V=800.0 PL=0
MOVL C01814 V=800.0 PL=0
MOVL C01815 V=800.0 PL=0
MOVL C01816 V=800.0 PL=0
MOVL C01817 V=800.0 PL=0
MOVL C01818 V=800.0 PL=0
MOVL C01819 V=800.0 PL=0
MOVL C01820 V=800.0 PL=0
MOVL C01821 V=800.0 PL=0
MOVL C01822 V=800.0 PL=0
MOVL C01823 V=800.0 PL=0
MOVL C01824 V=800.0 PL=0
MOVL C01825 V=800.0 PL=0
MOVL C01826 V=800.0 PL=0
MOVL C01827 V=800.0 PL=0
MOVL C01828 V=800.0 PL=0
MOVL C01829 V=800.0 PL=0
MOVL C01830 V=800.0 PL=0
MOVL C01831 V=800.0 PL=0
MOVL C01832 V=800.0 PL=0
MOVL C01833 V=800.0 PL=0
MOVL C01834 V=800.0 PL=0
MOVL C01835 V=800.0 PL=0
MOVL C01836 V=800.0 PL=0
MOVL C01837 V=800.0 PL=0
MOVL C01838 V=800.0 PL=0
MOVL C01839 V=800.0 PL=0
MOVL C01840 V=800.0 PL=0
MOVL C01841 V=800.0 PL=0
MOVL C01842 V=800.0 PL=0
MOVL C01843 V=800.0 PL=0
MOVL C01844 V=800.0 PL=0
MOVL C01845 V=800.0 PL=0
MOVL C01846 V=800.0 PL=0
MOVL C01847 V=800.0 PL=0
MOVL C01848 V=800.0 PL=0
MOVL C01849 V=800.0 PL=0
MOVL C01850 V=800.0 PL=0
MOVL C01851 V=800.0 PL=0
MOVL C01852 V=800.0 PL=0
MOVL C01853 V=800.0 PL=0
MOVL C01854 V=800.0 PL=0
MOVL C01855 V=800.0 PL=0
MOVL C01856 V=800.0 PL=0
MOVL C01857 V=800.0 PL=0
MOVL C01858 V=800.0 PL=0
MOVL C01859 V=800.0 PL=0
MOVL C01860 V=800.0 PL=0
MOVL C01861 V=800.0 PL=0
MOVL C01862 V=800.0 PL=0
MOVL C01863 V=800.0 PL=0
MOVL C01864 V=800.0 PL=0
MOVL C01865 V=800.0 PL=0
MOVL C01866 V=800.0 PL=0
MOVL C01867 V=800.0 PL=0
MOVL C01868 V=800.0 PL=0
MOVL C01869 V=800.0 PL=0
MOVL C01870 V=800.0 PL=0
MOVL C01871 V=800.0 PL=0
MOVL C01872 V=800.0 PL=0
MOVL C01873 V=800.0 PL=0
MOVL C01874 V=800.0 PL=0
MOVL C01875 V=800.0 PL=0
MOVL C01876 V=800.0 PL=0
MOVL C01877 V=800.0 PL=0
MOVL C01878 V=800.0 PL=0
MOVL C01879 V=800.0 PL=0
MOVL C01880 V=800.0 PL=0
MOVL C01881 V=800.0 PL=0
MOVL C01882 V=800.0 PL=0
MOVL C01883 V=800.0 PL=0
MOVL C01884 V=800.0 PL=0
MOVL C01885 V=800.0 PL=0
MOVL C01886 V=800.0 PL=0
MOVL C01887 V=800.0 PL=0
MOVL C01888 V=800.0 PL=0
MOVL C01889 V=800.0 PL=0
MOVL C01890 V=800.0 PL=0
MOVL C01891 V=800.0 PL=0
MOVL C01892 V=800.0 PL=0
MOVL C01893 V=800.0 PL=0
MOVL C01894 V=800.0 PL=0
MOVL C01895 V=800.0 PL=0
MOVL C01896 V=800.0 PL=0
MOVL C01897 V=800.0 PL=0
MOVL C01898 V=800.0 PL=0
MOVL C01899 V=800.0 PL=0
MOVL C01900 V=800.0 PL=0
MOVL C01901 V=800.0 PL=0
MOVL C01902 V=800.0 PL=0
MOVL C01903 V=800.0 PL=0
MOVL C01904 V=800.0 PL=0
MOVL C01905 V=800.0 PL=0
MOVL C01906 V=800.0 PL=0
MOVL C01907 V=800.0 PL=0
MOVL C01908 V=800.0 PL=0
MOVL C01909 V=800.0 PL=0
MOVL C01910 V=800.0 PL=0
MOVL C01911 V=800.0 PL=0
MOVL C01912 V=800.0 PL=0
MOVL C01913 V=800.0 PL=0
MOVL C01914 V=800.0 PL=0
MOVL C01915 V=800.0 PL=0
MOVL C01916 V=800.0 PL=0
MOVL C01917 V=800.0 PL=0
MOVL C01918 V=800.0 PL=0
MOVL C01919 V=800.0 PL=0
MOVL C01920 V=800.0 PL=0
MOVL C01921 V=800.0 PL=0
MOVL C01922 V=800.0 PL=0
MOVL C01923 V=800.0 PL=0
MOVL C01924 V=800.0 PL=0
MOVL C01925 V=800.0 PL=0
MOVL C01926 V=800.0 PL=0
MOVL C01927 V=800.0 PL=0
MOVL C01928 V=800.0 PL=0
MOVL C01929 V=800.0 PL=0
MOVL C01930 V=800.0 PL=0
MOVL C01931 V=800.0 PL=0
MOVL C01932 V=800.0 PL=0
MOVL C01933 V=800.0 PL=0
MOVL C01934 V=800.0 PL=0
MOVL C01935 V=800.0 PL=0
MOVL C01936 V=800.0 PL=0
MOVL C01937 V=800.0 PL=0
MOVL C01938 V=800.0 PL=0
MOVL C01939 V=800.0 PL=0
MOVL C01940 V=800.0 PL=0
MOVL C01941 V=800.0 PL=0
MOVL C01942 V=800.0 PL=0
MOVL C01943 V=800.0 PL=0
MOVL C01944 V=800.0 PL=0
MOVL C01945 V=800.0 PL=0
MOVL C01946 V=800.0 PL=0
MOVL C01947 V=800.0 PL=0
MOVL C01948 V=800.0 PL=0
MOVL C01949 V=800.0 PL=0
MOVL C01950 V=800.0 PL=0
MOVL C01951 V=800.0 PL=0
MOVL C01952 V=800.0 PL=0
MOVL C01953 V=800.0 PL=0
MOVL C01954 V=800.0 PL=0
MOVL C01955 V=800.0 PL=0
MOVL C01956 V=800.0 PL=0
MOVL C01957 V=800.0 PL=0
MOVL C01958 V=800.0 PL=0
MOVL C01959 V=800.0 PL=0
MOVL C01960 V=800.0 PL=0
MOVL C01961 V=800.0 PL=0
MOVL C01962 V=800.0 PL=0
MOVL C01963 V=800.0 PL=0
MOVL C01964 V=800.0 PL=0
MOVL C01965 V=800.0 PL=0
MOVL C01966 V=800.0 PL=0
MOVL C01967 V=800.0 PL=0
MOVL C01968 V=800.0 PL=0
MOVL C01969 V=800.0 PL=0
MOVL C01970 V=800.0 PL=0
MOVL C01971 V=800.0 PL=0
MOVL C01972 V=800.0 PL=0
MOVL C01973 V=800.0 PL=0
MOVL C01974 V=800.0 PL=0
MOVL C01975 V=800.0 PL=0
MOVL C01976 V=800.0 PL=0
MOVL C01977 V=800.0 PL=0
MOVL C01978 V=800.0 PL=0
MOVL C01979 V=800.0 PL=0
MOVL C01980 V=800.0 PL=0
MOVL C01981 V=800.0 PL=0
MOVL C01982 V=800.0 PL=0
MOVL C01983 V=800.0 PL=0
MOVL C01984 V=800.0 PL=0
MOVL C01985 V=800.0 PL=0
MOVL C01986 V=800.0 PL=0
MOVL C01987 V=800.0 PL=0
MOVL C01988 V=800.0 PL=0
MOVL C01989 V=800.0 PL=0
MOVL C01990 V=800.0 PL=0
MOVL C01991 V=800.0 PL=0
MOVL C01992 V=800.0 PL=0
MOVL C01993 V=800.0 PL=0
MOVL C01994 V=800.0 PL=0
MOVL C01995 V=800.0 PL=0
MOVL C01996 V=800.0 PL=0
MOVL C01997 V=800.0 PL=0
MOVL C01998 V=800.0 PL=0
MOVL C01999 V=800.0 PL=0
MOVL C02000 V=800.0 PL=0
MOVL C02001 V=800.0 PL=0
MOVL C02002 V=800.0 PL=0
MOVL C02003 V=800.0 PL=0
MOVL C02004 V=800.0 PL=0
MOVL C02005 V=800.0 PL=0
MOVL C02006 V=800.0 PL=0
MOVL C02007 V=800.0 PL=0
MOVL C02008 V=800.0 PL=0
MOVL C02009 V=800.0 PL=0
MOVL C02010 V=800.0 PL=0
MOVL C02011 V=800.0 PL=0
MOVL C02012 V=800.0 PL=0
MOVL C02013 V=800.0 PL=0
MOVL C02014 V=800.0 PL=0
MOVL C02015 V=800.0 PL=0
MOVL C02016 V=800.0 PL=0
MOVL C02017 V=800.0 PL=0
MOVL C02018 V=800.0 PL=0
MOVL C02019 V=800.0 PL=0
MOVL C02020 V=800.0 PL=0
MOVL C02021 V=800.0 PL=0
MOVL C02022 V=800.0 PL=0
MOVL C02023 V=800.0 PL=0
MOVL C02024 V=800.0 PL=0
MOVL C02025 V=800.0 PL=0
MOVL C02026 V=800.0 PL=0
MOVL C02027 V=800.0 PL=0
MOVL C02028 V=800.0 PL=0
MOVL C02029 V=800.0 PL=0
MOVL C02030 V=800.0 PL=0
MOVL C02031 V=800.0 PL=0
MOVL C02032 V=800.0 PL=0
MOVL C02033 V=800.0 PL=0
MOVL C02034 V=800.0 PL=0
MOVL C02035 V=800.0 PL=0
MOVL C02036 V=800.0 PL=0
MOVL C02037 V=800.0 PL=0
MOVL C02038 V=800.0 PL=0
MOVL C02039 V=800.0 PL=0
MOVL C02040 V=800.0 PL=0
MOVL C02041 V=800.0 PL=0
MOVL C02042 V=800.0 PL=0
MOVL C02043 V=800.0 PL=0
MOVL C02044 V=800.0 PL=0
MOVL C02045 V=800.0 PL=0
MOVL C02046 V=800.0 PL=0
MOVL C02047 V=800.0 PL=0
MOVL C02048 V=800.0 PL=0
MOVL C02049 V=800.0 PL=0
MOVL C02050 V=800.0 PL=0
MOVL C02051 V=800.0 PL=0
MOVL C02052 V=800.0 PL=0
MOVL C02053 V=800.0 PL=0
MOVL C02054 V=800.0 PL=0
MOVL C02055 V=800.0 PL=0
MOVL C02056 V=800.0 PL=0
MOVL C02057 V=800.0 PL=0
MOVL C02058 V=800.0 PL=0
MOVL C02059 V=800.0 PL=0
MOVL C02060 V=800.0 PL=0
MOVL C02061 V=800.0 PL=0
MOVL C02062 V=800.0 PL=0
MOVL C02063 V=800.0 PL=0
MOVL C02064 V=800.0 PL=0
MOVL C02065 V=800.0 PL=0
MOVL C02066 V=800.0 PL=0
MOVL C02067 V=800.0 PL=0
MOVL C02068 V=800.0 PL=0
MOVL C02069 V=800.0 PL=0
MOVL C02070 V=800.0 PL=0
MOVL C02071 V=800.0 PL=0
MOVL C02072 V=800.0 PL=0
MOVL C02073 V=800.0 PL=0
MOVL C02074 V=800.0 PL=0
MOVL C02075 V=800.0 PL=0
MOVL C02076 V=800.0 PL=0
MOVL C02077 V=800.0 PL=0
MOVL C02078 V=800.0 PL=0
MOVL C02079 V=800.0 PL=0
MOVL C02080 V=800.0 PL=0
MOVL C02081 V=800.0 PL=0
